   1:  PR[GP1:91,1] = PR[GP1:90,1] + 7.172;
   1:  PR[GP1:91,2] = PR[GP1:90,2] + -12.649;
   1:L PR[91] 10mm/sec CNT100;
   1:  PR[GP1:91,1] = PR[GP1:90,1] + 9.973;
   1:  PR[GP1:91,2] = PR[GP1:90,2] + -18.239;
   1:L PR[91] 10mm/sec CNT100;
   1:  PR[GP1:91,1] = PR[GP1:90,1] + 13.438;
   1:  PR[GP1:91,2] = PR[GP1:90,2] + -22.690;
   1:L PR[91] 10mm/sec CNT100;
   1:  PR[GP1:91,1] = PR[GP1:90,1] + 17.099;
   1:  PR[GP1:91,2] = PR[GP1:90,2] + -26.371;
   1:L PR[91] 10mm/sec CNT100;
   1:  PR[GP1:91,1] = PR[GP1:90,1] + 22.911;
   1:  PR[GP1:91,2] = PR[GP1:90,2] + -30.145;
   1:L PR[91] 10mm/sec CNT100;
   1:  PR[GP1:91,1] = PR[GP1:90,1] + 26.457;
   1:  PR[GP1:91,2] = PR[GP1:90,2] + -31.958;
   1:L PR[91] 10mm/sec CNT100;
   1:  PR[GP1:91,1] = PR[GP1:90,1] + 34.555;
   1:  PR[GP1:91,2] = PR[GP1:90,2] + -33.996;
   1:L PR[91] 10mm/sec CNT100;
   1:  PR[GP1:91,1] = PR[GP1:90,1] + 37.222;
   1:  PR[GP1:91,2] = PR[GP1:90,2] + -34.430;
   1:L PR[91] 10mm/sec CNT100;
   1:  PR[GP1:91,1] = PR[GP1:90,1] + 46.851;
   1:  PR[GP1:91,2] = PR[GP1:90,2] + -33.641;
   1:L PR[91] 10mm/sec CNT100;
   1:  PR[GP1:91,1] = PR[GP1:90,1] + 48.358;
   1:  PR[GP1:91,2] = PR[GP1:90,2] + -33.412;
   1:L PR[91] 10mm/sec CNT100;
   1:  PR[GP1:91,1] = PR[GP1:90,1] + 58.186;
   1:  PR[GP1:91,2] = PR[GP1:90,2] + -29.141;
   1:L PR[91] 10mm/sec CNT100;
   1:  PR[GP1:91,1] = PR[GP1:90,1] + 58.697;
   1:  PR[GP1:91,2] = PR[GP1:90,2] + -28.887;
   1:L PR[91] 10mm/sec CNT100;
   1:  PR[GP1:91,1] = PR[GP1:90,1] + 67.093;
   1:  PR[GP1:91,2] = PR[GP1:90,2] + -21.226;
   1:L PR[91] 10mm/sec CNT100;
   1:  PR[GP1:91,1] = PR[GP1:90,1] + 72.535;
   1:  PR[GP1:91,2] = PR[GP1:90,2] + -11.242;
   1:L PR[91] 10mm/sec CNT100;
   1:  PR[GP1:91,1] = PR[GP1:90,1] + 72.559;
   1:  PR[GP1:91,2] = PR[GP1:90,2] + -11.160;
   1:L PR[91] 10mm/sec CNT100;
   1:  PR[GP1:91,1] = PR[GP1:90,1] + 72.575;
   1:  PR[GP1:91,2] = PR[GP1:90,2] + -10.988;
   1:L PR[91] 10mm/sec CNT100;
   1:  PR[GP1:91,1] = PR[GP1:90,1] + 74.410;
   1:  PR[GP1:91,2] = PR[GP1:90,2] + 0.017;
   1:L PR[91] 10mm/sec CNT100;
   1:  PR[GP1:91,1] = PR[GP1:90,1] + 74.379;
   1:  PR[GP1:91,2] = PR[GP1:90,2] + 0.350;
   1:L PR[91] 10mm/sec CNT100;
   1:  PR[GP1:91,1] = PR[GP1:90,1] + 72.565;
   1:  PR[GP1:91,2] = PR[GP1:90,2] + 11.130;
   1:L PR[91] 10mm/sec CNT100;
   1:  PR[GP1:91,1] = PR[GP1:90,1] + 72.535;
   1:  PR[GP1:91,2] = PR[GP1:90,2] + 11.234;
   1:L PR[91] 10mm/sec CNT100;
   1:  PR[GP1:91,1] = PR[GP1:90,1] + 67.091;
   1:  PR[GP1:91,2] = PR[GP1:90,2] + 21.219;
   1:L PR[91] 10mm/sec CNT100;
   1:  PR[GP1:91,1] = PR[GP1:90,1] + 58.697;
   1:  PR[GP1:91,2] = PR[GP1:90,2] + 28.878;
   1:L PR[91] 10mm/sec CNT100;
   1:  PR[GP1:91,1] = PR[GP1:90,1] + 58.186;
   1:  PR[GP1:91,2] = PR[GP1:90,2] + 29.133;
   1:L PR[91] 10mm/sec CNT100;
   1:  PR[GP1:91,1] = PR[GP1:90,1] + 48.358;
   1:  PR[GP1:91,2] = PR[GP1:90,2] + 33.403;
   1:L PR[91] 10mm/sec CNT100;
   1:  PR[GP1:91,1] = PR[GP1:90,1] + 46.851;
   1:  PR[GP1:91,2] = PR[GP1:90,2] + 33.632;
   1:L PR[91] 10mm/sec CNT100;
   1:  PR[GP1:91,1] = PR[GP1:90,1] + 37.222;
   1:  PR[GP1:91,2] = PR[GP1:90,2] + 34.421;
   1:L PR[91] 10mm/sec CNT100;
   1:  PR[GP1:91,1] = PR[GP1:90,1] + 34.555;
   1:  PR[GP1:91,2] = PR[GP1:90,2] + 33.987;
   1:L PR[91] 10mm/sec CNT100;
   1:  PR[GP1:91,1] = PR[GP1:90,1] + 26.457;
   1:  PR[GP1:91,2] = PR[GP1:90,2] + 31.949;
   1:L PR[91] 10mm/sec CNT100;
   1:  PR[GP1:91,1] = PR[GP1:90,1] + 22.911;
   1:  PR[GP1:91,2] = PR[GP1:90,2] + 30.136;
   1:L PR[91] 10mm/sec CNT100;
   1:  PR[GP1:91,1] = PR[GP1:90,1] + 17.099;
   1:  PR[GP1:91,2] = PR[GP1:90,2] + 26.362;
   1:L PR[91] 10mm/sec CNT100;
   1:  PR[GP1:91,1] = PR[GP1:90,1] + 13.438;
   1:  PR[GP1:91,2] = PR[GP1:90,2] + 22.681;
   1:L PR[91] 10mm/sec CNT100;
   1:  PR[GP1:91,1] = PR[GP1:90,1] + 9.973;
   1:  PR[GP1:91,2] = PR[GP1:90,2] + 18.230;
   1:L PR[91] 10mm/sec CNT100;
   1:  PR[GP1:91,1] = PR[GP1:90,1] + 7.168;
   1:  PR[GP1:91,2] = PR[GP1:90,2] + 12.628;
   1:L PR[91] 10mm/sec CNT100;
   1:  PR[GP1:91,1] = PR[GP1:90,1] + 5.691;
   1:  PR[GP1:91,2] = PR[GP1:90,2] + 8.281;
   1:L PR[91] 10mm/sec CNT100;
   1:  PR[GP1:91,1] = PR[GP1:90,1] + 5.052;
   1:  PR[GP1:91,2] = PR[GP1:90,2] + 6.468;
   1:L PR[91] 10mm/sec CNT100;
   1:  PR[GP1:91,1] = PR[GP1:90,1] + 4.191;
   1:  PR[GP1:91,2] = PR[GP1:90,2] + 5.426;
   1:L PR[91] 10mm/sec CNT100;
   1:  PR[GP1:91,1] = PR[GP1:90,1] + 2.887;
   1:  PR[GP1:91,2] = PR[GP1:90,2] + 4.007;
   1:L PR[91] 10mm/sec CNT100;
   1:  PR[GP1:91,1] = PR[GP1:90,1] + 2.240;
   1:  PR[GP1:91,2] = PR[GP1:90,2] + 3.649;
   1:L PR[91] 10mm/sec CNT100;
   1:  PR[GP1:91,1] = PR[GP1:90,1] + 0.884;
   1:  PR[GP1:91,2] = PR[GP1:90,2] + 4.821;
   1:  PR[GP1:91,3] = PR[GP1:90,3] + 21.280;
   1:L PR[91] 10mm/sec CNT100;
   1:  PR[GP1:91,1] = PR[GP1:90,1] + -1.866;
   1:  PR[GP1:91,2] = PR[GP1:90,2] + 5.029;
   1:L PR[91] 10mm/sec CNT100;
   1:  PR[GP1:91,1] = PR[GP1:90,1] + -2.248;
   1:  PR[GP1:91,2] = PR[GP1:90,2] + 5.297;
   1:L PR[91] 10mm/sec CNT100;
   1:  PR[GP1:91,1] = PR[GP1:90,1] + -3.405;
   1:  PR[GP1:91,2] = PR[GP1:90,2] + 6.715;
   1:L PR[91] 10mm/sec CNT100;
   1:  PR[GP1:91,1] = PR[GP1:90,1] + -4.805;
   1:  PR[GP1:91,2] = PR[GP1:90,2] + 9.191;
   1:L PR[91] 10mm/sec CNT100;
   1:  PR[GP1:91,1] = PR[GP1:90,1] + -5.571;
   1:  PR[GP1:91,2] = PR[GP1:90,2] + 11.449;
   1:L PR[91] 10mm/sec CNT100;
   1:  PR[GP1:91,1] = PR[GP1:90,1] + -9.332;
   1:  PR[GP1:91,2] = PR[GP1:90,2] + 18.969;
   1:L PR[91] 10mm/sec CNT100;
   1:  PR[GP1:91,1] = PR[GP1:90,1] + -11.484;
   1:  PR[GP1:91,2] = PR[GP1:90,2] + 21.732;
   1:L PR[91] 10mm/sec CNT100;
   1:  PR[GP1:91,1] = PR[GP1:90,1] + -16.563;
   1:  PR[GP1:91,2] = PR[GP1:90,2] + 26.824;
   1:L PR[91] 10mm/sec CNT100;
   1:  PR[GP1:91,1] = PR[GP1:90,1] + -20.680;
   1:  PR[GP1:91,2] = PR[GP1:90,2] + 29.498;
   1:L PR[91] 10mm/sec CNT100;
   1:  PR[GP1:91,1] = PR[GP1:90,1] + -25.923;
   1:  PR[GP1:91,2] = PR[GP1:90,2] + 32.179;
   1:L PR[91] 10mm/sec CNT100;
   1:  PR[GP1:91,1] = PR[GP1:90,1] + -32.191;
   1:  PR[GP1:91,2] = PR[GP1:90,2] + 33.756;
   1:L PR[91] 10mm/sec CNT100;
   1:  PR[GP1:91,1] = PR[GP1:90,1] + -36.623;
   1:  PR[GP1:91,2] = PR[GP1:90,2] + 34.474;
   1:L PR[91] 10mm/sec CNT100;
   1:  PR[GP1:91,1] = PR[GP1:90,1] + -44.511;
   1:  PR[GP1:91,2] = PR[GP1:90,2] + 33.827;
   1:L PR[91] 10mm/sec CNT100;
   1:  PR[GP1:91,1] = PR[GP1:90,1] + -47.660;
   1:  PR[GP1:91,2] = PR[GP1:90,2] + 33.349;
   1:L PR[91] 10mm/sec CNT100;
   1:  PR[GP1:91,1] = PR[GP1:90,1] + -56.007;
   1:  PR[GP1:91,2] = PR[GP1:90,2] + 29.720;
   1:L PR[91] 10mm/sec CNT100;
   1:  PR[GP1:91,1] = PR[GP1:90,1] + -57.896;
   1:  PR[GP1:91,2] = PR[GP1:90,2] + 28.777;
   1:L PR[91] 10mm/sec CNT100;
   1:  PR[GP1:91,1] = PR[GP1:90,1] + -65.248;
   1:  PR[GP1:91,2] = PR[GP1:90,2] + 22.071;
   1:L PR[91] 10mm/sec CNT100;
   1:  PR[GP1:91,1] = PR[GP1:90,1] + -66.199;
   1:  PR[GP1:91,2] = PR[GP1:90,2] + 21.135;
   1:L PR[91] 10mm/sec CNT100;
   1:  PR[GP1:91,1] = PR[GP1:90,1] + -71.212;
   1:  PR[GP1:91,2] = PR[GP1:90,2] + 11.956;
   1:L PR[91] 10mm/sec CNT100;
   1:  PR[GP1:91,1] = PR[GP1:90,1] + -71.611;
   1:  PR[GP1:91,2] = PR[GP1:90,2] + 11.183;
   1:L PR[91] 10mm/sec CNT100;
   1:  PR[GP1:91,1] = PR[GP1:90,1] + -73.500;
   1:  PR[GP1:91,2] = PR[GP1:90,2] + -0.004;
   1:L PR[91] 10mm/sec CNT100;
   1:  PR[GP1:91,1] = PR[GP1:90,1] + -71.736;
   1:  PR[GP1:91,2] = PR[GP1:90,2] + -10.406;
   1:L PR[91] 10mm/sec CNT100;
   1:  PR[GP1:91,1] = PR[GP1:90,1] + -71.610;
   1:  PR[GP1:91,2] = PR[GP1:90,2] + -11.194;
   1:L PR[91] 10mm/sec CNT100;
   1:  PR[GP1:91,1] = PR[GP1:90,1] + -71.212;
   1:  PR[GP1:91,2] = PR[GP1:90,2] + -11.965;
   1:L PR[91] 10mm/sec CNT100;
   1:  PR[GP1:91,1] = PR[GP1:90,1] + -66.199;
   1:  PR[GP1:91,2] = PR[GP1:90,2] + -21.144;
   1:L PR[91] 10mm/sec CNT100;
   1:  PR[GP1:91,1] = PR[GP1:90,1] + -65.248;
   1:  PR[GP1:91,2] = PR[GP1:90,2] + -22.080;
   1:L PR[91] 10mm/sec CNT100;
   1:  PR[GP1:91,1] = PR[GP1:90,1] + -57.896;
   1:  PR[GP1:91,2] = PR[GP1:90,2] + -28.786;
   1:L PR[91] 10mm/sec CNT100;
   1:  PR[GP1:91,1] = PR[GP1:90,1] + -56.007;
   1:  PR[GP1:91,2] = PR[GP1:90,2] + -29.729;
   1:L PR[91] 10mm/sec CNT100;
   1:  PR[GP1:91,1] = PR[GP1:90,1] + -47.660;
   1:  PR[GP1:91,2] = PR[GP1:90,2] + -33.358;
   1:L PR[91] 10mm/sec CNT100;
   1:  PR[GP1:91,1] = PR[GP1:90,1] + -44.511;
   1:  PR[GP1:91,2] = PR[GP1:90,2] + -33.836;
   1:L PR[91] 10mm/sec CNT100;
   1:  PR[GP1:91,1] = PR[GP1:90,1] + -36.623;
   1:  PR[GP1:91,2] = PR[GP1:90,2] + -34.483;
   1:L PR[91] 10mm/sec CNT100;
   1:  PR[GP1:91,1] = PR[GP1:90,1] + -32.191;
   1:  PR[GP1:91,2] = PR[GP1:90,2] + -33.765;
   1:L PR[91] 10mm/sec CNT100;
   1:  PR[GP1:91,1] = PR[GP1:90,1] + -25.924;
   1:  PR[GP1:91,2] = PR[GP1:90,2] + -32.188;
   1:L PR[91] 10mm/sec CNT100;
   1:  PR[GP1:91,1] = PR[GP1:90,1] + -20.680;
   1:  PR[GP1:91,2] = PR[GP1:90,2] + -29.507;
   1:L PR[91] 10mm/sec CNT100;
   1:  PR[GP1:91,1] = PR[GP1:90,1] + -16.563;
   1:  PR[GP1:91,2] = PR[GP1:90,2] + -26.833;
   1:L PR[91] 10mm/sec CNT100;
   1:  PR[GP1:91,1] = PR[GP1:90,1] + -11.484;
   1:  PR[GP1:91,2] = PR[GP1:90,2] + -21.741;
   1:L PR[91] 10mm/sec CNT100;
   1:  PR[GP1:91,1] = PR[GP1:90,1] + -9.332;
   1:  PR[GP1:91,2] = PR[GP1:90,2] + -18.977;
   1:L PR[91] 10mm/sec CNT100;
   1:  PR[GP1:91,1] = PR[GP1:90,1] + -5.576;
   1:  PR[GP1:91,2] = PR[GP1:90,2] + -11.474;
   1:L PR[91] 10mm/sec CNT100;
   1:  PR[GP1:91,1] = PR[GP1:90,1] + -4.308;
   1:  PR[GP1:91,2] = PR[GP1:90,2] + -7.786;
   1:L PR[91] 10mm/sec CNT100;
   1:  PR[GP1:91,1] = PR[GP1:90,1] + -3.131;
   1:  PR[GP1:91,2] = PR[GP1:90,2] + -6.484;
   1:L PR[91] 10mm/sec CNT100;
   1:  PR[GP1:91,1] = PR[GP1:90,1] + -2.802;
   1:  PR[GP1:91,2] = PR[GP1:90,2] + -6.283;
   1:L PR[91] 10mm/sec CNT100;
   1:  PR[GP1:91,1] = PR[GP1:90,1] + -1.567;
   1:  PR[GP1:91,2] = PR[GP1:90,2] + -4.807;
   1:L PR[91] 10mm/sec CNT100;
   1:  PR[GP1:91,1] = PR[GP1:90,1] + 1.456;
   1:  PR[GP1:91,2] = PR[GP1:90,2] + -5.040;
   1:L PR[91] 10mm/sec CNT100;
   1:  PR[GP1:91,1] = PR[GP1:90,1] + 1.588;
   1:  PR[GP1:91,2] = PR[GP1:90,2] + -5.147;
   1:L PR[91] 10mm/sec CNT100;
   1:  PR[GP1:91,1] = PR[GP1:90,1] + 2.989;
   1:  PR[GP1:91,2] = PR[GP1:90,2] + -5.133;
   1:L PR[91] 10mm/sec CNT100;
   1:  PR[GP1:91,1] = PR[GP1:90,1] + 4.319;
   1:  PR[GP1:91,2] = PR[GP1:90,2] + -7.663;
   1:L PR[91] 10mm/sec CNT100;
   1:  PR[GP1:91,1] = PR[GP1:90,1] + 5.601;
   1:  PR[GP1:91,2] = PR[GP1:90,2] + -9.140;
   1:L PR[91] 10mm/sec CNT100;
   1:  PR[GP1:91,1] = PR[GP1:90,1] + 6.392;
   1:  PR[GP1:91,2] = PR[GP1:90,2] + -11.470;
   1:L PR[91] 10mm/sec CNT100;
   1:  PR[GP1:91,1] = PR[GP1:90,1] + 10.145;
   1:  PR[GP1:91,2] = PR[GP1:90,2] + -18.959;
   1:L PR[91] 10mm/sec CNT100;
   1:  PR[GP1:91,1] = PR[GP1:90,1] + 12.297;
   1:  PR[GP1:91,2] = PR[GP1:90,2] + -21.723;
   1:L PR[91] 10mm/sec CNT100;
   1:  PR[GP1:91,1] = PR[GP1:90,1] + 17.376;
   1:  PR[GP1:91,2] = PR[GP1:90,2] + -26.830;
   1:L PR[91] 10mm/sec CNT100;
   1:  PR[GP1:91,1] = PR[GP1:90,1] + 21.491;
   1:  PR[GP1:91,2] = PR[GP1:90,2] + -29.502;
   1:L PR[91] 10mm/sec CNT100;
   1:  PR[GP1:91,1] = PR[GP1:90,1] + 26.737;
   1:  PR[GP1:91,2] = PR[GP1:90,2] + -32.185;
   1:L PR[91] 10mm/sec CNT100;
   1:  PR[GP1:91,1] = PR[GP1:90,1] + 33.004;
   1:  PR[GP1:91,2] = PR[GP1:90,2] + -33.762;
   1:L PR[91] 10mm/sec CNT100;
   1:  PR[GP1:91,1] = PR[GP1:90,1] + 37.438;
   1:  PR[GP1:91,2] = PR[GP1:90,2] + -34.483;
   1:L PR[91] 10mm/sec CNT100;
   1:  PR[GP1:91,1] = PR[GP1:90,1] + 45.326;
   1:  PR[GP1:91,2] = PR[GP1:90,2] + -33.836;
   1:L PR[91] 10mm/sec CNT100;
   1:  PR[GP1:91,1] = PR[GP1:90,1] + 48.477;
   1:  PR[GP1:91,2] = PR[GP1:90,2] + -33.358;
   1:L PR[91] 10mm/sec CNT100;
   1:  PR[GP1:91,1] = PR[GP1:90,1] + 56.825;
   1:  PR[GP1:91,2] = PR[GP1:90,2] + -29.731;
   1:L PR[91] 10mm/sec CNT100;
   1:  PR[GP1:91,1] = PR[GP1:90,1] + 58.715;
   1:  PR[GP1:91,2] = PR[GP1:90,2] + -28.789;
   1:L PR[91] 10mm/sec CNT100;
   1:  PR[GP1:91,1] = PR[GP1:90,1] + 66.067;
   1:  PR[GP1:91,2] = PR[GP1:90,2] + -22.080;
   1:L PR[91] 10mm/sec CNT100;
   1:  PR[GP1:91,1] = PR[GP1:90,1] + 67.019;
   1:  PR[GP1:91,2] = PR[GP1:90,2] + -21.142;
   1:L PR[91] 10mm/sec CNT100;
   1:  PR[GP1:91,1] = PR[GP1:90,1] + 72.032;
   1:  PR[GP1:91,2] = PR[GP1:90,2] + -11.969;
   1:L PR[91] 10mm/sec CNT100;
   1:  PR[GP1:91,1] = PR[GP1:90,1] + 72.432;
   1:  PR[GP1:91,2] = PR[GP1:90,2] + -11.197;
   1:L PR[91] 10mm/sec CNT100;
   1:  PR[GP1:91,1] = PR[GP1:90,1] + 74.321;
   1:  PR[GP1:91,2] = PR[GP1:90,2] + -0.004;
   1:L PR[91] 10mm/sec CNT100;
   1:  PR[GP1:91,1] = PR[GP1:90,1] + 72.432;
   1:  PR[GP1:91,2] = PR[GP1:90,2] + 11.188;
   1:L PR[91] 10mm/sec CNT100;
   1:  PR[GP1:91,1] = PR[GP1:90,1] + 72.032;
   1:  PR[GP1:91,2] = PR[GP1:90,2] + 11.960;
   1:L PR[91] 10mm/sec CNT100;
   1:  PR[GP1:91,1] = PR[GP1:90,1] + 67.019;
   1:  PR[GP1:91,2] = PR[GP1:90,2] + 21.133;
   1:L PR[91] 10mm/sec CNT100;
   1:  PR[GP1:91,1] = PR[GP1:90,1] + 66.067;
   1:  PR[GP1:91,2] = PR[GP1:90,2] + 22.071;
   1:L PR[91] 10mm/sec CNT100;
   1:  PR[GP1:91,1] = PR[GP1:90,1] + 58.715;
   1:  PR[GP1:91,2] = PR[GP1:90,2] + 28.780;
   1:L PR[91] 10mm/sec CNT100;
   1:  PR[GP1:91,1] = PR[GP1:90,1] + 56.825;
   1:  PR[GP1:91,2] = PR[GP1:90,2] + 29.722;
   1:L PR[91] 10mm/sec CNT100;
   1:  PR[GP1:91,1] = PR[GP1:90,1] + 48.477;
   1:  PR[GP1:91,2] = PR[GP1:90,2] + 33.349;
   1:L PR[91] 10mm/sec CNT100;
   1:  PR[GP1:91,1] = PR[GP1:90,1] + 45.326;
   1:  PR[GP1:91,2] = PR[GP1:90,2] + 33.828;
   1:L PR[91] 10mm/sec CNT100;
   1:  PR[GP1:91,1] = PR[GP1:90,1] + 37.438;
   1:  PR[GP1:91,2] = PR[GP1:90,2] + 34.474;
   1:L PR[91] 10mm/sec CNT100;
   1:  PR[GP1:91,1] = PR[GP1:90,1] + 33.004;
   1:  PR[GP1:91,2] = PR[GP1:90,2] + 33.753;
   1:L PR[91] 10mm/sec CNT100;
   1:  PR[GP1:91,1] = PR[GP1:90,1] + 26.737;
   1:  PR[GP1:91,2] = PR[GP1:90,2] + 32.176;
   1:L PR[91] 10mm/sec CNT100;
   1:  PR[GP1:91,1] = PR[GP1:90,1] + 21.491;
   1:  PR[GP1:91,2] = PR[GP1:90,2] + 29.494;
   1:L PR[91] 10mm/sec CNT100;
   1:  PR[GP1:91,1] = PR[GP1:90,1] + 17.375;
   1:  PR[GP1:91,2] = PR[GP1:90,2] + 26.821;
   1:L PR[91] 10mm/sec CNT100;
   1:  PR[GP1:91,1] = PR[GP1:90,1] + 12.297;
   1:  PR[GP1:91,2] = PR[GP1:90,2] + 21.714;
   1:L PR[91] 10mm/sec CNT100;
   1:  PR[GP1:91,1] = PR[GP1:90,1] + 10.145;
   1:  PR[GP1:91,2] = PR[GP1:90,2] + 18.950;
   1:L PR[91] 10mm/sec CNT100;
   1:  PR[GP1:91,1] = PR[GP1:90,1] + 6.385;
   1:  PR[GP1:91,2] = PR[GP1:90,2] + 11.443;
   1:L PR[91] 10mm/sec CNT100;
   1:  PR[GP1:91,1] = PR[GP1:90,1] + 5.125;
   1:  PR[GP1:91,2] = PR[GP1:90,2] + 7.774;
   1:L PR[91] 10mm/sec CNT100;
   1:  PR[GP1:91,1] = PR[GP1:90,1] + 3.922;
   1:  PR[GP1:91,2] = PR[GP1:90,2] + 6.317;
   1:L PR[91] 10mm/sec CNT100;
   1:  PR[GP1:91,1] = PR[GP1:90,1] + 2.826;
   1:  PR[GP1:91,2] = PR[GP1:90,2] + 5.125;
   1:L PR[91] 10mm/sec CNT100;
   1:  PR[GP1:91,1] = PR[GP1:90,1] + 2.251;
   1:  PR[GP1:91,2] = PR[GP1:90,2] + 4.806;
   1:L PR[91] 10mm/sec CNT100;
   1:  PR[GP1:91,1] = PR[GP1:90,1] + 0.410;
   1:  PR[GP1:91,2] = PR[GP1:90,2] + 5.983;
   1:  PR[GP1:91,3] = PR[GP1:90,3] + 22.610;
   1:L PR[91] 10mm/sec CNT100;
   1:  PR[GP1:91,1] = PR[GP1:90,1] + -1.815;
   1:  PR[GP1:91,2] = PR[GP1:90,2] + 6.152;
   1:L PR[91] 10mm/sec CNT100;
   1:  PR[GP1:91,1] = PR[GP1:90,1] + -2.161;
   1:  PR[GP1:91,2] = PR[GP1:90,2] + 6.394;
   1:L PR[91] 10mm/sec CNT100;
   1:  PR[GP1:91,1] = PR[GP1:90,1] + -3.724;
   1:  PR[GP1:91,2] = PR[GP1:90,2] + 8.310;
   1:L PR[91] 10mm/sec CNT100;
   1:  PR[GP1:91,1] = PR[GP1:90,1] + -4.752;
   1:  PR[GP1:91,2] = PR[GP1:90,2] + 10.152;
   1:L PR[91] 10mm/sec CNT100;
   1:  PR[GP1:91,1] = PR[GP1:90,1] + -4.791;
   1:  PR[GP1:91,2] = PR[GP1:90,2] + 10.265;
   1:L PR[91] 10mm/sec CNT100;
   1:  PR[GP1:91,1] = PR[GP1:90,1] + -9.505;
   1:  PR[GP1:91,2] = PR[GP1:90,2] + 19.692;
   1:L PR[91] 10mm/sec CNT100;
   1:  PR[GP1:91,1] = PR[GP1:90,1] + -10.345;
   1:  PR[GP1:91,2] = PR[GP1:90,2] + 20.769;
   1:L PR[91] 10mm/sec CNT100;
   1:  PR[GP1:91,1] = PR[GP1:90,1] + -16.841;
   1:  PR[GP1:91,2] = PR[GP1:90,2] + 27.284;
   1:L PR[91] 10mm/sec CNT100;
   1:  PR[GP1:91,1] = PR[GP1:90,1] + -19.262;
   1:  PR[GP1:91,2] = PR[GP1:90,2] + 28.856;
   1:L PR[91] 10mm/sec CNT100;
   1:  PR[GP1:91,1] = PR[GP1:90,1] + -26.205;
   1:  PR[GP1:91,2] = PR[GP1:90,2] + 32.407;
   1:L PR[91] 10mm/sec CNT100;
   1:  PR[GP1:91,1] = PR[GP1:90,1] + -30.643;
   1:  PR[GP1:91,2] = PR[GP1:90,2] + 33.523;
   1:L PR[91] 10mm/sec CNT100;
   1:  PR[GP1:91,1] = PR[GP1:90,1] + -36.840;
   1:  PR[GP1:91,2] = PR[GP1:90,2] + 34.527;
   1:L PR[91] 10mm/sec CNT100;
   1:  PR[GP1:91,1] = PR[GP1:90,1] + -42.988;
   1:  PR[GP1:91,2] = PR[GP1:90,2] + 34.023;
   1:L PR[91] 10mm/sec CNT100;
   1:  PR[GP1:91,1] = PR[GP1:90,1] + -47.779;
   1:  PR[GP1:91,2] = PR[GP1:90,2] + 33.295;
   1:L PR[91] 10mm/sec CNT100;
   1:  PR[GP1:91,1] = PR[GP1:90,1] + -54.648;
   1:  PR[GP1:91,2] = PR[GP1:90,2] + 30.310;
   1:L PR[91] 10mm/sec CNT100;
   1:  PR[GP1:91,1] = PR[GP1:90,1] + -57.914;
   1:  PR[GP1:91,2] = PR[GP1:90,2] + 28.679;
   1:L PR[91] 10mm/sec CNT100;
   1:  PR[GP1:91,1] = PR[GP1:90,1] + -64.160;
   1:  PR[GP1:91,2] = PR[GP1:90,2] + 22.982;
   1:L PR[91] 10mm/sec CNT100;
   1:  PR[GP1:91,1] = PR[GP1:90,1] + -66.132;
   1:  PR[GP1:91,2] = PR[GP1:90,2] + 21.041;
   1:L PR[91] 10mm/sec CNT100;
   1:  PR[GP1:91,1] = PR[GP1:90,1] + -70.470;
   1:  PR[GP1:91,2] = PR[GP1:90,2] + 13.096;
   1:L PR[91] 10mm/sec CNT100;
   1:  PR[GP1:91,1] = PR[GP1:90,1] + -71.488;
   1:  PR[GP1:91,2] = PR[GP1:90,2] + 11.127;
   1:L PR[91] 10mm/sec CNT100;
   1:  PR[GP1:91,1] = PR[GP1:90,1] + -73.081;
   1:  PR[GP1:91,2] = PR[GP1:90,2] + 1.714;
   1:L PR[91] 10mm/sec CNT100;
   1:  PR[GP1:91,1] = PR[GP1:90,1] + -73.356;
   1:  PR[GP1:91,2] = PR[GP1:90,2] + -0.002;
   1:L PR[91] 10mm/sec CNT100;
   1:  PR[GP1:91,1] = PR[GP1:90,1] + -71.808;
   1:  PR[GP1:91,2] = PR[GP1:90,2] + -9.130;
   1:L PR[91] 10mm/sec CNT100;
   1:  PR[GP1:91,1] = PR[GP1:90,1] + -71.486;
   1:  PR[GP1:91,2] = PR[GP1:90,2] + -11.139;
   1:L PR[91] 10mm/sec CNT100;
   1:  PR[GP1:91,1] = PR[GP1:90,1] + -70.470;
   1:  PR[GP1:91,2] = PR[GP1:90,2] + -13.105;
   1:L PR[91] 10mm/sec CNT100;
   1:  PR[GP1:91,1] = PR[GP1:90,1] + -66.132;
   1:  PR[GP1:91,2] = PR[GP1:90,2] + -21.050;
   1:L PR[91] 10mm/sec CNT100;
   1:  PR[GP1:91,1] = PR[GP1:90,1] + -64.159;
   1:  PR[GP1:91,2] = PR[GP1:90,2] + -22.991;
   1:L PR[91] 10mm/sec CNT100;
   1:  PR[GP1:91,1] = PR[GP1:90,1] + -57.914;
   1:  PR[GP1:91,2] = PR[GP1:90,2] + -28.688;
   1:L PR[91] 10mm/sec CNT100;
   1:  PR[GP1:91,1] = PR[GP1:90,1] + -54.648;
   1:  PR[GP1:91,2] = PR[GP1:90,2] + -30.319;
   1:L PR[91] 10mm/sec CNT100;
   1:  PR[GP1:91,1] = PR[GP1:90,1] + -47.779;
   1:  PR[GP1:91,2] = PR[GP1:90,2] + -33.304;
   1:L PR[91] 10mm/sec CNT100;
   1:  PR[GP1:91,1] = PR[GP1:90,1] + -42.988;
   1:  PR[GP1:91,2] = PR[GP1:90,2] + -34.032;
   1:L PR[91] 10mm/sec CNT100;
   1:  PR[GP1:91,1] = PR[GP1:90,1] + -36.840;
   1:  PR[GP1:91,2] = PR[GP1:90,2] + -34.536;
   1:L PR[91] 10mm/sec CNT100;
   1:  PR[GP1:91,1] = PR[GP1:90,1] + -30.643;
   1:  PR[GP1:91,2] = PR[GP1:90,2] + -33.532;
   1:L PR[91] 10mm/sec CNT100;
   1:  PR[GP1:91,1] = PR[GP1:90,1] + -26.205;
   1:  PR[GP1:91,2] = PR[GP1:90,2] + -32.415;
   1:L PR[91] 10mm/sec CNT100;
   1:  PR[GP1:91,1] = PR[GP1:90,1] + -19.262;
   1:  PR[GP1:91,2] = PR[GP1:90,2] + -28.865;
   1:L PR[91] 10mm/sec CNT100;
   1:  PR[GP1:91,1] = PR[GP1:90,1] + -16.841;
   1:  PR[GP1:91,2] = PR[GP1:90,2] + -27.293;
   1:L PR[91] 10mm/sec CNT100;
   1:  PR[GP1:91,1] = PR[GP1:90,1] + -10.345;
   1:  PR[GP1:91,2] = PR[GP1:90,2] + -20.778;
   1:L PR[91] 10mm/sec CNT100;
   1:  PR[GP1:91,1] = PR[GP1:90,1] + -9.505;
   1:  PR[GP1:91,2] = PR[GP1:90,2] + -19.701;
   1:L PR[91] 10mm/sec CNT100;
   1:  PR[GP1:91,1] = PR[GP1:90,1] + -4.797;
   1:  PR[GP1:91,2] = PR[GP1:90,2] + -10.293;
   1:L PR[91] 10mm/sec CNT100;
   1:  PR[GP1:91,1] = PR[GP1:90,1] + -4.382;
   1:  PR[GP1:91,2] = PR[GP1:90,2] + -9.094;
   1:L PR[91] 10mm/sec CNT100;
   1:  PR[GP1:91,1] = PR[GP1:90,1] + -3.503;
   1:  PR[GP1:91,2] = PR[GP1:90,2] + -8.122;
   1:L PR[91] 10mm/sec CNT100;
   1:  PR[GP1:91,1] = PR[GP1:90,1] + -3.272;
   1:  PR[GP1:91,2] = PR[GP1:90,2] + -7.981;
   1:L PR[91] 10mm/sec CNT100;
   1:  PR[GP1:91,1] = PR[GP1:90,1] + -1.588;
   1:  PR[GP1:91,2] = PR[GP1:90,2] + -5.970;
   1:L PR[91] 10mm/sec CNT100;
   1:  PR[GP1:91,1] = PR[GP1:90,1] + 0.917;
   1:  PR[GP1:91,2] = PR[GP1:90,2] + -6.163;
   1:L PR[91] 10mm/sec CNT100;
   1:  PR[GP1:91,1] = PR[GP1:90,1] + 1.018;
   1:  PR[GP1:91,2] = PR[GP1:90,2] + -6.244;
   1:L PR[91] 10mm/sec CNT100;
   1:  PR[GP1:91,1] = PR[GP1:90,1] + 2.892;
   1:  PR[GP1:91,2] = PR[GP1:90,2] + -6.225;
   1:L PR[91] 10mm/sec CNT100;
   1:  PR[GP1:91,1] = PR[GP1:90,1] + 3.978;
   1:  PR[GP1:91,2] = PR[GP1:90,2] + -8.293;
   1:L PR[91] 10mm/sec CNT100;
   1:  PR[GP1:91,1] = PR[GP1:90,1] + 5.547;
   1:  PR[GP1:91,2] = PR[GP1:90,2] + -10.099;
   1:L PR[91] 10mm/sec CNT100;
   1:  PR[GP1:91,1] = PR[GP1:90,1] + 5.611;
   1:  PR[GP1:91,2] = PR[GP1:90,2] + -10.290;
   1:L PR[91] 10mm/sec CNT100;
   1:  PR[GP1:91,1] = PR[GP1:90,1] + 10.317;
   1:  PR[GP1:91,2] = PR[GP1:90,2] + -19.679;
   1:L PR[91] 10mm/sec CNT100;
   1:  PR[GP1:91,1] = PR[GP1:90,1] + 11.155;
   1:  PR[GP1:91,2] = PR[GP1:90,2] + -20.756;
   1:L PR[91] 10mm/sec CNT100;
   1:  PR[GP1:91,1] = PR[GP1:90,1] + 17.652;
   1:  PR[GP1:91,2] = PR[GP1:90,2] + -27.289;
   1:L PR[91] 10mm/sec CNT100;
   1:  PR[GP1:91,1] = PR[GP1:90,1] + 20.071;
   1:  PR[GP1:91,2] = PR[GP1:90,2] + -28.860;
   1:L PR[91] 10mm/sec CNT100;
   1:  PR[GP1:91,1] = PR[GP1:90,1] + 27.017;
   1:  PR[GP1:91,2] = PR[GP1:90,2] + -32.411;
   1:L PR[91] 10mm/sec CNT100;
   1:  PR[GP1:91,1] = PR[GP1:90,1] + 31.454;
   1:  PR[GP1:91,2] = PR[GP1:90,2] + -33.528;
   1:L PR[91] 10mm/sec CNT100;
   1:  PR[GP1:91,1] = PR[GP1:90,1] + 37.654;
   1:  PR[GP1:91,2] = PR[GP1:90,2] + -34.536;
   1:L PR[91] 10mm/sec CNT100;
   1:  PR[GP1:91,1] = PR[GP1:90,1] + 43.802;
   1:  PR[GP1:91,2] = PR[GP1:90,2] + -34.032;
   1:L PR[91] 10mm/sec CNT100;
   1:  PR[GP1:91,1] = PR[GP1:90,1] + 48.596;
   1:  PR[GP1:91,2] = PR[GP1:90,2] + -33.305;
   1:L PR[91] 10mm/sec CNT100;
   1:  PR[GP1:91,1] = PR[GP1:90,1] + 55.464;
   1:  PR[GP1:91,2] = PR[GP1:90,2] + -30.320;
   1:L PR[91] 10mm/sec CNT100;
   1:  PR[GP1:91,1] = PR[GP1:90,1] + 58.732;
   1:  PR[GP1:91,2] = PR[GP1:90,2] + -28.691;
   1:L PR[91] 10mm/sec CNT100;
   1:  PR[GP1:91,1] = PR[GP1:90,1] + 64.978;
   1:  PR[GP1:91,2] = PR[GP1:90,2] + -22.992;
   1:L PR[91] 10mm/sec CNT100;
   1:  PR[GP1:91,1] = PR[GP1:90,1] + 66.951;
   1:  PR[GP1:91,2] = PR[GP1:90,2] + -21.047;
   1:L PR[91] 10mm/sec CNT100;
   1:  PR[GP1:91,1] = PR[GP1:90,1] + 71.290;
   1:  PR[GP1:91,2] = PR[GP1:90,2] + -13.107;
   1:L PR[91] 10mm/sec CNT100;
   1:  PR[GP1:91,1] = PR[GP1:90,1] + 72.308;
   1:  PR[GP1:91,2] = PR[GP1:90,2] + -11.143;
   1:L PR[91] 10mm/sec CNT100;
   1:  PR[GP1:91,1] = PR[GP1:90,1] + 73.902;
   1:  PR[GP1:91,2] = PR[GP1:90,2] + -1.725;
   1:L PR[91] 10mm/sec CNT100;
   1:  PR[GP1:91,1] = PR[GP1:90,1] + 74.177;
   1:  PR[GP1:91,2] = PR[GP1:90,2] + -0.007;
   1:L PR[91] 10mm/sec CNT100;
   1:  PR[GP1:91,1] = PR[GP1:90,1] + 72.628;
   1:  PR[GP1:91,2] = PR[GP1:90,2] + 9.125;
   1:L PR[91] 10mm/sec CNT100;
   1:  PR[GP1:91,1] = PR[GP1:90,1] + 72.307;
   1:  PR[GP1:91,2] = PR[GP1:90,2] + 11.137;
   1:L PR[91] 10mm/sec CNT100;
   1:  PR[GP1:91,1] = PR[GP1:90,1] + 71.290;
   1:  PR[GP1:91,2] = PR[GP1:90,2] + 13.099;
   1:L PR[91] 10mm/sec CNT100;
   1:  PR[GP1:91,1] = PR[GP1:90,1] + 66.951;
   1:  PR[GP1:91,2] = PR[GP1:90,2] + 21.038;
   1:L PR[91] 10mm/sec CNT100;
   1:  PR[GP1:91,1] = PR[GP1:90,1] + 64.978;
   1:  PR[GP1:91,2] = PR[GP1:90,2] + 22.983;
   1:L PR[91] 10mm/sec CNT100;
   1:  PR[GP1:91,1] = PR[GP1:90,1] + 58.732;
   1:  PR[GP1:91,2] = PR[GP1:90,2] + 28.682;
   1:L PR[91] 10mm/sec CNT100;
   1:  PR[GP1:91,1] = PR[GP1:90,1] + 55.464;
   1:  PR[GP1:91,2] = PR[GP1:90,2] + 30.311;
   1:L PR[91] 10mm/sec CNT100;
   1:  PR[GP1:91,1] = PR[GP1:90,1] + 48.596;
   1:  PR[GP1:91,2] = PR[GP1:90,2] + 33.296;
   1:L PR[91] 10mm/sec CNT100;
   1:  PR[GP1:91,1] = PR[GP1:90,1] + 43.802;
   1:  PR[GP1:91,2] = PR[GP1:90,2] + 34.023;
   1:L PR[91] 10mm/sec CNT100;
   1:  PR[GP1:91,1] = PR[GP1:90,1] + 37.654;
   1:  PR[GP1:91,2] = PR[GP1:90,2] + 34.527;
   1:L PR[91] 10mm/sec CNT100;
   1:  PR[GP1:91,1] = PR[GP1:90,1] + 31.454;
   1:  PR[GP1:91,2] = PR[GP1:90,2] + 33.519;
   1:L PR[91] 10mm/sec CNT100;
   1:  PR[GP1:91,1] = PR[GP1:90,1] + 27.017;
   1:  PR[GP1:91,2] = PR[GP1:90,2] + 32.402;
   1:L PR[91] 10mm/sec CNT100;
   1:  PR[GP1:91,1] = PR[GP1:90,1] + 20.071;
   1:  PR[GP1:91,2] = PR[GP1:90,2] + 28.851;
   1:L PR[91] 10mm/sec CNT100;
   1:  PR[GP1:91,1] = PR[GP1:90,1] + 17.652;
   1:  PR[GP1:91,2] = PR[GP1:90,2] + 27.280;
   1:L PR[91] 10mm/sec CNT100;
   1:  PR[GP1:91,1] = PR[GP1:90,1] + 11.155;
   1:  PR[GP1:91,2] = PR[GP1:90,2] + 20.747;
   1:L PR[91] 10mm/sec CNT100;
   1:  PR[GP1:91,1] = PR[GP1:90,1] + 10.317;
   1:  PR[GP1:91,2] = PR[GP1:90,2] + 19.670;
   1:L PR[91] 10mm/sec CNT100;
   1:  PR[GP1:91,1] = PR[GP1:90,1] + 5.604;
   1:  PR[GP1:91,2] = PR[GP1:90,2] + 10.259;
   1:L PR[91] 10mm/sec CNT100;
   1:  PR[GP1:91,1] = PR[GP1:90,1] + 5.196;
   1:  PR[GP1:91,2] = PR[GP1:90,2] + 9.078;
   1:L PR[91] 10mm/sec CNT100;
   1:  PR[GP1:91,1] = PR[GP1:90,1] + 3.653;
   1:  PR[GP1:91,2] = PR[GP1:90,2] + 7.209;
   1:L PR[91] 10mm/sec CNT100;
   1:  PR[GP1:91,1] = PR[GP1:90,1] + 2.765;
   1:  PR[GP1:91,2] = PR[GP1:90,2] + 6.242;
   1:L PR[91] 10mm/sec CNT100;
   1:  PR[GP1:91,1] = PR[GP1:90,1] + 2.261;
   1:  PR[GP1:91,2] = PR[GP1:90,2] + 5.964;
   1:L PR[91] 10mm/sec CNT100;
   1:  PR[GP1:91,1] = PR[GP1:90,1] + -0.065;
   1:  PR[GP1:91,2] = PR[GP1:90,2] + 7.146;
   1:  PR[GP1:91,3] = PR[GP1:90,3] + 23.940;
   1:L PR[91] 10mm/sec CNT100;
   1:  PR[GP1:91,1] = PR[GP1:90,1] + -1.765;
   1:  PR[GP1:91,2] = PR[GP1:90,2] + 7.274;
   1:L PR[91] 10mm/sec CNT100;
   1:  PR[GP1:91,1] = PR[GP1:90,1] + -2.074;
   1:  PR[GP1:91,2] = PR[GP1:90,2] + 7.491;
   1:L PR[91] 10mm/sec CNT100;
   1:  PR[GP1:91,1] = PR[GP1:90,1] + -4.043;
   1:  PR[GP1:91,2] = PR[GP1:90,2] + 9.904;
   1:L PR[91] 10mm/sec CNT100;
   1:  PR[GP1:91,1] = PR[GP1:90,1] + -4.665;
   1:  PR[GP1:91,2] = PR[GP1:90,2] + 11.023;
   1:L PR[91] 10mm/sec CNT100;
   1:  PR[GP1:91,1] = PR[GP1:90,1] + -9.277;
   1:  PR[GP1:91,2] = PR[GP1:90,2] + 19.846;
   1:L PR[91] 10mm/sec CNT100;
   1:  PR[GP1:91,1] = PR[GP1:90,1] + -9.604;
   1:  PR[GP1:91,2] = PR[GP1:90,2] + 20.320;
   1:L PR[91] 10mm/sec CNT100;
   1:  PR[GP1:91,1] = PR[GP1:90,1] + -12.636;
   1:  PR[GP1:91,2] = PR[GP1:90,2] + 23.248;
   1:L PR[91] 10mm/sec CNT100;
   1:  PR[GP1:91,1] = PR[GP1:90,1] + -17.120;
   1:  PR[GP1:91,2] = PR[GP1:90,2] + 27.744;
   1:L PR[91] 10mm/sec CNT100;
   1:  PR[GP1:91,1] = PR[GP1:90,1] + -17.844;
   1:  PR[GP1:91,2] = PR[GP1:90,2] + 28.215;
   1:L PR[91] 10mm/sec CNT100;
   1:  PR[GP1:91,1] = PR[GP1:90,1] + -26.487;
   1:  PR[GP1:91,2] = PR[GP1:90,2] + 32.634;
   1:L PR[91] 10mm/sec CNT100;
   1:  PR[GP1:91,1] = PR[GP1:90,1] + -29.094;
   1:  PR[GP1:91,2] = PR[GP1:90,2] + 33.290;
   1:L PR[91] 10mm/sec CNT100;
   1:  PR[GP1:91,1] = PR[GP1:90,1] + -37.057;
   1:  PR[GP1:91,2] = PR[GP1:90,2] + 34.580;
   1:L PR[91] 10mm/sec CNT100;
   1:  PR[GP1:91,1] = PR[GP1:90,1] + -41.465;
   1:  PR[GP1:91,2] = PR[GP1:90,2] + 34.219;
   1:L PR[91] 10mm/sec CNT100;
   1:  PR[GP1:91,1] = PR[GP1:90,1] + -47.899;
   1:  PR[GP1:91,2] = PR[GP1:90,2] + 33.242;
   1:L PR[91] 10mm/sec CNT100;
   1:  PR[GP1:91,1] = PR[GP1:90,1] + -53.288;
   1:  PR[GP1:91,2] = PR[GP1:90,2] + 30.899;
   1:L PR[91] 10mm/sec CNT100;
   1:  PR[GP1:91,1] = PR[GP1:90,1] + -57.932;
   1:  PR[GP1:91,2] = PR[GP1:90,2] + 28.580;
   1:L PR[91] 10mm/sec CNT100;
   1:  PR[GP1:91,1] = PR[GP1:90,1] + -63.071;
   1:  PR[GP1:91,2] = PR[GP1:90,2] + 23.893;
   1:L PR[91] 10mm/sec CNT100;
   1:  PR[GP1:91,1] = PR[GP1:90,1] + -66.064;
   1:  PR[GP1:91,2] = PR[GP1:90,2] + 20.947;
   1:L PR[91] 10mm/sec CNT100;
   1:  PR[GP1:91,1] = PR[GP1:90,1] + -69.728;
   1:  PR[GP1:91,2] = PR[GP1:90,2] + 14.236;
   1:L PR[91] 10mm/sec CNT100;
   1:  PR[GP1:91,1] = PR[GP1:90,1] + -71.364;
   1:  PR[GP1:91,2] = PR[GP1:90,2] + 11.072;
   1:L PR[91] 10mm/sec CNT100;
   1:  PR[GP1:91,1] = PR[GP1:90,1] + -72.728;
   1:  PR[GP1:91,2] = PR[GP1:90,2] + 3.014;
   1:L PR[91] 10mm/sec CNT100;
   1:  PR[GP1:91,1] = PR[GP1:90,1] + -73.211;
   1:  PR[GP1:91,2] = PR[GP1:90,2] + -0.002;
   1:L PR[91] 10mm/sec CNT100;
   1:  PR[GP1:91,1] = PR[GP1:90,1] + -71.879;
   1:  PR[GP1:91,2] = PR[GP1:90,2] + -7.854;
   1:L PR[91] 10mm/sec CNT100;
   1:  PR[GP1:91,1] = PR[GP1:90,1] + -71.362;
   1:  PR[GP1:91,2] = PR[GP1:90,2] + -11.083;
   1:L PR[91] 10mm/sec CNT100;
   1:  PR[GP1:91,1] = PR[GP1:90,1] + -69.728;
   1:  PR[GP1:91,2] = PR[GP1:90,2] + -14.245;
   1:L PR[91] 10mm/sec CNT100;
   1:  PR[GP1:91,1] = PR[GP1:90,1] + -66.064;
   1:  PR[GP1:91,2] = PR[GP1:90,2] + -20.956;
   1:L PR[91] 10mm/sec CNT100;
   1:  PR[GP1:91,1] = PR[GP1:90,1] + -63.071;
   1:  PR[GP1:91,2] = PR[GP1:90,2] + -23.902;
   1:L PR[91] 10mm/sec CNT100;
   1:  PR[GP1:91,1] = PR[GP1:90,1] + -57.932;
   1:  PR[GP1:91,2] = PR[GP1:90,2] + -28.589;
   1:L PR[91] 10mm/sec CNT100;
   1:  PR[GP1:91,1] = PR[GP1:90,1] + -53.288;
   1:  PR[GP1:91,2] = PR[GP1:90,2] + -30.908;
   1:L PR[91] 10mm/sec CNT100;
   1:  PR[GP1:91,1] = PR[GP1:90,1] + -47.899;
   1:  PR[GP1:91,2] = PR[GP1:90,2] + -33.251;
   1:L PR[91] 10mm/sec CNT100;
   1:  PR[GP1:91,1] = PR[GP1:90,1] + -41.465;
   1:  PR[GP1:91,2] = PR[GP1:90,2] + -34.228;
   1:L PR[91] 10mm/sec CNT100;
   1:  PR[GP1:91,1] = PR[GP1:90,1] + -37.057;
   1:  PR[GP1:91,2] = PR[GP1:90,2] + -34.589;
   1:L PR[91] 10mm/sec CNT100;
   1:  PR[GP1:91,1] = PR[GP1:90,1] + -29.094;
   1:  PR[GP1:91,2] = PR[GP1:90,2] + -33.298;
   1:L PR[91] 10mm/sec CNT100;
   1:  PR[GP1:91,1] = PR[GP1:90,1] + -26.487;
   1:  PR[GP1:91,2] = PR[GP1:90,2] + -32.643;
   1:L PR[91] 10mm/sec CNT100;
   1:  PR[GP1:91,1] = PR[GP1:90,1] + -17.844;
   1:  PR[GP1:91,2] = PR[GP1:90,2] + -28.224;
   1:L PR[91] 10mm/sec CNT100;
   1:  PR[GP1:91,1] = PR[GP1:90,1] + -17.120;
   1:  PR[GP1:91,2] = PR[GP1:90,2] + -27.753;
   1:L PR[91] 10mm/sec CNT100;
   1:  PR[GP1:91,1] = PR[GP1:90,1] + -12.636;
   1:  PR[GP1:91,2] = PR[GP1:90,2] + -23.257;
   1:L PR[91] 10mm/sec CNT100;
   1:  PR[GP1:91,1] = PR[GP1:90,1] + -9.604;
   1:  PR[GP1:91,2] = PR[GP1:90,2] + -20.329;
   1:L PR[91] 10mm/sec CNT100;
   1:  PR[GP1:91,1] = PR[GP1:90,1] + -9.275;
   1:  PR[GP1:91,2] = PR[GP1:90,2] + -19.852;
   1:L PR[91] 10mm/sec CNT100;
   1:  PR[GP1:91,1] = PR[GP1:90,1] + -4.689;
   1:  PR[GP1:91,2] = PR[GP1:90,2] + -11.079;
   1:L PR[91] 10mm/sec CNT100;
   1:  PR[GP1:91,1] = PR[GP1:90,1] + -4.456;
   1:  PR[GP1:91,2] = PR[GP1:90,2] + -10.403;
   1:L PR[91] 10mm/sec CNT100;
   1:  PR[GP1:91,1] = PR[GP1:90,1] + -3.875;
   1:  PR[GP1:91,2] = PR[GP1:90,2] + -9.761;
   1:L PR[91] 10mm/sec CNT100;
   1:  PR[GP1:91,1] = PR[GP1:90,1] + -3.742;
   1:  PR[GP1:91,2] = PR[GP1:90,2] + -9.679;
   1:L PR[91] 10mm/sec CNT100;
   1:  PR[GP1:91,1] = PR[GP1:90,1] + -1.610;
   1:  PR[GP1:91,2] = PR[GP1:90,2] + -7.132;
   1:L PR[91] 10mm/sec CNT100;
   1:  PR[GP1:91,1] = PR[GP1:90,1] + 0.379;
   1:  PR[GP1:91,2] = PR[GP1:90,2] + -7.285;
   1:L PR[91] 10mm/sec CNT100;
   1:  PR[GP1:91,1] = PR[GP1:90,1] + 0.448;
   1:  PR[GP1:91,2] = PR[GP1:90,2] + -7.341;
   1:L PR[91] 10mm/sec CNT100;
   1:  PR[GP1:91,1] = PR[GP1:90,1] + 2.794;
   1:  PR[GP1:91,2] = PR[GP1:90,2] + -7.317;
   1:L PR[91] 10mm/sec CNT100;
   1:  PR[GP1:91,1] = PR[GP1:90,1] + 3.638;
   1:  PR[GP1:91,2] = PR[GP1:90,2] + -8.922;
   1:L PR[91] 10mm/sec CNT100;
   1:  PR[GP1:91,1] = PR[GP1:90,1] + 4.759;
   1:  PR[GP1:91,2] = PR[GP1:90,2] + -10.213;
   1:L PR[91] 10mm/sec CNT100;
   1:  PR[GP1:91,1] = PR[GP1:90,1] + 5.446;
   1:  PR[GP1:91,2] = PR[GP1:90,2] + -10.966;
   1:L PR[91] 10mm/sec CNT100;
   1:  PR[GP1:91,1] = PR[GP1:90,1] + 10.085;
   1:  PR[GP1:91,2] = PR[GP1:90,2] + -19.826;
   1:L PR[91] 10mm/sec CNT100;
   1:  PR[GP1:91,1] = PR[GP1:90,1] + 10.415;
   1:  PR[GP1:91,2] = PR[GP1:90,2] + -20.306;
   1:L PR[91] 10mm/sec CNT100;
   1:  PR[GP1:91,1] = PR[GP1:90,1] + 13.457;
   1:  PR[GP1:91,2] = PR[GP1:90,2] + -23.251;
   1:L PR[91] 10mm/sec CNT100;
   1:  PR[GP1:91,1] = PR[GP1:90,1] + 17.929;
   1:  PR[GP1:91,2] = PR[GP1:90,2] + -27.748;
   1:L PR[91] 10mm/sec CNT100;
   1:  PR[GP1:91,1] = PR[GP1:90,1] + 18.652;
   1:  PR[GP1:91,2] = PR[GP1:90,2] + -28.217;
   1:L PR[91] 10mm/sec CNT100;
   1:  PR[GP1:91,1] = PR[GP1:90,1] + 27.297;
   1:  PR[GP1:91,2] = PR[GP1:90,2] + -32.638;
   1:L PR[91] 10mm/sec CNT100;
   1:  PR[GP1:91,1] = PR[GP1:90,1] + 29.903;
   1:  PR[GP1:91,2] = PR[GP1:90,2] + -33.293;
   1:L PR[91] 10mm/sec CNT100;
   1:  PR[GP1:91,1] = PR[GP1:90,1] + 37.870;
   1:  PR[GP1:91,2] = PR[GP1:90,2] + -34.589;
   1:L PR[91] 10mm/sec CNT100;
   1:  PR[GP1:91,1] = PR[GP1:90,1] + 42.277;
   1:  PR[GP1:91,2] = PR[GP1:90,2] + -34.228;
   1:L PR[91] 10mm/sec CNT100;
   1:  PR[GP1:91,1] = PR[GP1:90,1] + 48.714;
   1:  PR[GP1:91,2] = PR[GP1:90,2] + -33.251;
   1:L PR[91] 10mm/sec CNT100;
   1:  PR[GP1:91,1] = PR[GP1:90,1] + 54.104;
   1:  PR[GP1:91,2] = PR[GP1:90,2] + -30.909;
   1:L PR[91] 10mm/sec CNT100;
   1:  PR[GP1:91,1] = PR[GP1:90,1] + 58.749;
   1:  PR[GP1:91,2] = PR[GP1:90,2] + -28.593;
   1:L PR[91] 10mm/sec CNT100;
   1:  PR[GP1:91,1] = PR[GP1:90,1] + 63.888;
   1:  PR[GP1:91,2] = PR[GP1:90,2] + -23.904;
   1:L PR[91] 10mm/sec CNT100;
   1:  PR[GP1:91,1] = PR[GP1:90,1] + 66.884;
   1:  PR[GP1:91,2] = PR[GP1:90,2] + -20.953;
   1:L PR[91] 10mm/sec CNT100;
   1:  PR[GP1:91,1] = PR[GP1:90,1] + 70.548;
   1:  PR[GP1:91,2] = PR[GP1:90,2] + -14.246;
   1:L PR[91] 10mm/sec CNT100;
   1:  PR[GP1:91,1] = PR[GP1:90,1] + 72.184;
   1:  PR[GP1:91,2] = PR[GP1:90,2] + -11.090;
   1:L PR[91] 10mm/sec CNT100;
   1:  PR[GP1:91,1] = PR[GP1:90,1] + 73.548;
   1:  PR[GP1:91,2] = PR[GP1:90,2] + -3.028;
   1:L PR[91] 10mm/sec CNT100;
   1:  PR[GP1:91,1] = PR[GP1:90,1] + 74.032;
   1:  PR[GP1:91,2] = PR[GP1:90,2] + -0.007;
   1:L PR[91] 10mm/sec CNT100;
   1:  PR[GP1:91,1] = PR[GP1:90,1] + 72.700;
   1:  PR[GP1:91,2] = PR[GP1:90,2] + 7.849;
   1:L PR[91] 10mm/sec CNT100;
   1:  PR[GP1:91,1] = PR[GP1:90,1] + 72.183;
   1:  PR[GP1:91,2] = PR[GP1:90,2] + 11.083;
   1:L PR[91] 10mm/sec CNT100;
   1:  PR[GP1:91,1] = PR[GP1:90,1] + 70.548;
   1:  PR[GP1:91,2] = PR[GP1:90,2] + 14.238;
   1:L PR[91] 10mm/sec CNT100;
   1:  PR[GP1:91,1] = PR[GP1:90,1] + 66.883;
   1:  PR[GP1:91,2] = PR[GP1:90,2] + 20.944;
   1:L PR[91] 10mm/sec CNT100;
   1:  PR[GP1:91,1] = PR[GP1:90,1] + 63.888;
   1:  PR[GP1:91,2] = PR[GP1:90,2] + 23.895;
   1:L PR[91] 10mm/sec CNT100;
   1:  PR[GP1:91,1] = PR[GP1:90,1] + 58.749;
   1:  PR[GP1:91,2] = PR[GP1:90,2] + 28.584;
   1:L PR[91] 10mm/sec CNT100;
   1:  PR[GP1:91,1] = PR[GP1:90,1] + 54.104;
   1:  PR[GP1:91,2] = PR[GP1:90,2] + 30.900;
   1:L PR[91] 10mm/sec CNT100;
   1:  PR[GP1:91,1] = PR[GP1:90,1] + 48.714;
   1:  PR[GP1:91,2] = PR[GP1:90,2] + 33.242;
   1:L PR[91] 10mm/sec CNT100;
   1:  PR[GP1:91,1] = PR[GP1:90,1] + 42.277;
   1:  PR[GP1:91,2] = PR[GP1:90,2] + 34.219;
   1:L PR[91] 10mm/sec CNT100;
   1:  PR[GP1:91,1] = PR[GP1:90,1] + 37.870;
   1:  PR[GP1:91,2] = PR[GP1:90,2] + 34.581;
   1:L PR[91] 10mm/sec CNT100;
   1:  PR[GP1:91,1] = PR[GP1:90,1] + 29.903;
   1:  PR[GP1:91,2] = PR[GP1:90,2] + 33.284;
   1:L PR[91] 10mm/sec CNT100;
   1:  PR[GP1:91,1] = PR[GP1:90,1] + 27.297;
   1:  PR[GP1:91,2] = PR[GP1:90,2] + 32.629;
   1:L PR[91] 10mm/sec CNT100;
   1:  PR[GP1:91,1] = PR[GP1:90,1] + 18.651;
   1:  PR[GP1:91,2] = PR[GP1:90,2] + 28.208;
   1:L PR[91] 10mm/sec CNT100;
   1:  PR[GP1:91,1] = PR[GP1:90,1] + 17.929;
   1:  PR[GP1:91,2] = PR[GP1:90,2] + 27.739;
   1:L PR[91] 10mm/sec CNT100;
   1:  PR[GP1:91,1] = PR[GP1:90,1] + 13.457;
   1:  PR[GP1:91,2] = PR[GP1:90,2] + 23.242;
   1:L PR[91] 10mm/sec CNT100;
   1:  PR[GP1:91,1] = PR[GP1:90,1] + 10.415;
   1:  PR[GP1:91,2] = PR[GP1:90,2] + 20.297;
   1:L PR[91] 10mm/sec CNT100;
   1:  PR[GP1:91,1] = PR[GP1:90,1] + 10.086;
   1:  PR[GP1:91,2] = PR[GP1:90,2] + 19.820;
   1:L PR[91] 10mm/sec CNT100;
   1:  PR[GP1:91,1] = PR[GP1:90,1] + 5.503;
   1:  PR[GP1:91,2] = PR[GP1:90,2] + 11.066;
   1:L PR[91] 10mm/sec CNT100;
   1:  PR[GP1:91,1] = PR[GP1:90,1] + 5.268;
   1:  PR[GP1:91,2] = PR[GP1:90,2] + 10.382;
   1:L PR[91] 10mm/sec CNT100;
   1:  PR[GP1:91,1] = PR[GP1:90,1] + 3.384;
   1:  PR[GP1:91,2] = PR[GP1:90,2] + 8.100;
   1:L PR[91] 10mm/sec CNT100;
   1:  PR[GP1:91,1] = PR[GP1:90,1] + 2.704;
   1:  PR[GP1:91,2] = PR[GP1:90,2] + 7.360;
   1:L PR[91] 10mm/sec CNT100;
   1:  PR[GP1:91,1] = PR[GP1:90,1] + 2.272;
   1:  PR[GP1:91,2] = PR[GP1:90,2] + 7.121;
   1:L PR[91] 10mm/sec CNT100;
   1:  PR[GP1:91,1] = PR[GP1:90,1] + -0.539;
   1:  PR[GP1:91,2] = PR[GP1:90,2] + 8.308;
   1:  PR[GP1:91,3] = PR[GP1:90,3] + 25.270;
   1:L PR[91] 10mm/sec CNT100;
   1:  PR[GP1:91,1] = PR[GP1:90,1] + -1.715;
   1:  PR[GP1:91,2] = PR[GP1:90,2] + 8.397;
   1:L PR[91] 10mm/sec CNT100;
   1:  PR[GP1:91,1] = PR[GP1:90,1] + -1.987;
   1:  PR[GP1:91,2] = PR[GP1:90,2] + 8.588;
   1:L PR[91] 10mm/sec CNT100;
   1:  PR[GP1:91,1] = PR[GP1:90,1] + -4.361;
   1:  PR[GP1:91,2] = PR[GP1:90,2] + 11.497;
   1:L PR[91] 10mm/sec CNT100;
   1:  PR[GP1:91,1] = PR[GP1:90,1] + -4.598;
   1:  PR[GP1:91,2] = PR[GP1:90,2] + 11.923;
   1:L PR[91] 10mm/sec CNT100;
   1:  PR[GP1:91,1] = PR[GP1:90,1] + -8.162;
   1:  PR[GP1:91,2] = PR[GP1:90,2] + 18.729;
   1:L PR[91] 10mm/sec CNT100;
   1:  PR[GP1:91,1] = PR[GP1:90,1] + -9.700;
   1:  PR[GP1:91,2] = PR[GP1:90,2] + 20.957;
   1:L PR[91] 10mm/sec CNT100;
   1:  PR[GP1:91,1] = PR[GP1:90,1] + -16.516;
   1:  PR[GP1:91,2] = PR[GP1:90,2] + 27.540;
   1:L PR[91] 10mm/sec CNT100;
   1:  PR[GP1:91,1] = PR[GP1:90,1] + -17.274;
   1:  PR[GP1:91,2] = PR[GP1:90,2] + 28.125;
   1:L PR[91] 10mm/sec CNT100;
   1:  PR[GP1:91,1] = PR[GP1:90,1] + -22.301;
   1:  PR[GP1:91,2] = PR[GP1:90,2] + 30.577;
   1:L PR[91] 10mm/sec CNT100;
   1:  PR[GP1:91,1] = PR[GP1:90,1] + -26.768;
   1:  PR[GP1:91,2] = PR[GP1:90,2] + 32.861;
   1:L PR[91] 10mm/sec CNT100;
   1:  PR[GP1:91,1] = PR[GP1:90,1] + -27.546;
   1:  PR[GP1:91,2] = PR[GP1:90,2] + 33.057;
   1:L PR[91] 10mm/sec CNT100;
   1:  PR[GP1:91,1] = PR[GP1:90,1] + -37.274;
   1:  PR[GP1:91,2] = PR[GP1:90,2] + 34.634;
   1:L PR[91] 10mm/sec CNT100;
   1:  PR[GP1:91,1] = PR[GP1:90,1] + -39.942;
   1:  PR[GP1:91,2] = PR[GP1:90,2] + 34.415;
   1:L PR[91] 10mm/sec CNT100;
   1:  PR[GP1:91,1] = PR[GP1:90,1] + -48.019;
   1:  PR[GP1:91,2] = PR[GP1:90,2] + 33.188;
   1:L PR[91] 10mm/sec CNT100;
   1:  PR[GP1:91,1] = PR[GP1:90,1] + -51.929;
   1:  PR[GP1:91,2] = PR[GP1:90,2] + 31.488;
   1:L PR[91] 10mm/sec CNT100;
   1:  PR[GP1:91,1] = PR[GP1:90,1] + -57.950;
   1:  PR[GP1:91,2] = PR[GP1:90,2] + 28.481;
   1:L PR[91] 10mm/sec CNT100;
   1:  PR[GP1:91,1] = PR[GP1:90,1] + -61.982;
   1:  PR[GP1:91,2] = PR[GP1:90,2] + 24.804;
   1:L PR[91] 10mm/sec CNT100;
   1:  PR[GP1:91,1] = PR[GP1:90,1] + -65.997;
   1:  PR[GP1:91,2] = PR[GP1:90,2] + 20.853;
   1:L PR[91] 10mm/sec CNT100;
   1:  PR[GP1:91,1] = PR[GP1:90,1] + -68.987;
   1:  PR[GP1:91,2] = PR[GP1:90,2] + 15.377;
   1:L PR[91] 10mm/sec CNT100;
   1:  PR[GP1:91,1] = PR[GP1:90,1] + -71.240;
   1:  PR[GP1:91,2] = PR[GP1:90,2] + 11.017;
   1:L PR[91] 10mm/sec CNT100;
   1:  PR[GP1:91,1] = PR[GP1:90,1] + -72.374;
   1:  PR[GP1:91,2] = PR[GP1:90,2] + 4.314;
   1:L PR[91] 10mm/sec CNT100;
   1:  PR[GP1:91,1] = PR[GP1:90,1] + -73.066;
   1:  PR[GP1:91,2] = PR[GP1:90,2] + -0.002;
   1:L PR[91] 10mm/sec CNT100;
   1:  PR[GP1:91,1] = PR[GP1:90,1] + -71.951;
   1:  PR[GP1:91,2] = PR[GP1:90,2] + -6.579;
   1:L PR[91] 10mm/sec CNT100;
   1:  PR[GP1:91,1] = PR[GP1:90,1] + -71.239;
   1:  PR[GP1:91,2] = PR[GP1:90,2] + -11.028;
   1:L PR[91] 10mm/sec CNT100;
   1:  PR[GP1:91,1] = PR[GP1:90,1] + -68.987;
   1:  PR[GP1:91,2] = PR[GP1:90,2] + -15.385;
   1:L PR[91] 10mm/sec CNT100;
   1:  PR[GP1:91,1] = PR[GP1:90,1] + -65.997;
   1:  PR[GP1:91,2] = PR[GP1:90,2] + -20.861;
   1:L PR[91] 10mm/sec CNT100;
   1:  PR[GP1:91,1] = PR[GP1:90,1] + -61.982;
   1:  PR[GP1:91,2] = PR[GP1:90,2] + -24.812;
   1:L PR[91] 10mm/sec CNT100;
   1:  PR[GP1:91,1] = PR[GP1:90,1] + -57.950;
   1:  PR[GP1:91,2] = PR[GP1:90,2] + -28.490;
   1:L PR[91] 10mm/sec CNT100;
   1:  PR[GP1:91,1] = PR[GP1:90,1] + -51.929;
   1:  PR[GP1:91,2] = PR[GP1:90,2] + -31.497;
   1:L PR[91] 10mm/sec CNT100;
   1:  PR[GP1:91,1] = PR[GP1:90,1] + -48.019;
   1:  PR[GP1:91,2] = PR[GP1:90,2] + -33.197;
   1:L PR[91] 10mm/sec CNT100;
   1:  PR[GP1:91,1] = PR[GP1:90,1] + -39.942;
   1:  PR[GP1:91,2] = PR[GP1:90,2] + -34.424;
   1:L PR[91] 10mm/sec CNT100;
   1:  PR[GP1:91,1] = PR[GP1:90,1] + -37.274;
   1:  PR[GP1:91,2] = PR[GP1:90,2] + -34.642;
   1:L PR[91] 10mm/sec CNT100;
   1:  PR[GP1:91,1] = PR[GP1:90,1] + -27.546;
   1:  PR[GP1:91,2] = PR[GP1:90,2] + -33.065;
   1:L PR[91] 10mm/sec CNT100;
   1:  PR[GP1:91,1] = PR[GP1:90,1] + -26.768;
   1:  PR[GP1:91,2] = PR[GP1:90,2] + -32.870;
   1:L PR[91] 10mm/sec CNT100;
   1:  PR[GP1:91,1] = PR[GP1:90,1] + -22.301;
   1:  PR[GP1:91,2] = PR[GP1:90,2] + -30.585;
   1:L PR[91] 10mm/sec CNT100;
   1:  PR[GP1:91,1] = PR[GP1:90,1] + -17.274;
   1:  PR[GP1:91,2] = PR[GP1:90,2] + -28.134;
   1:L PR[91] 10mm/sec CNT100;
   1:  PR[GP1:91,1] = PR[GP1:90,1] + -16.516;
   1:  PR[GP1:91,2] = PR[GP1:90,2] + -27.549;
   1:L PR[91] 10mm/sec CNT100;
   1:  PR[GP1:91,1] = PR[GP1:90,1] + -9.700;
   1:  PR[GP1:91,2] = PR[GP1:90,2] + -20.966;
   1:L PR[91] 10mm/sec CNT100;
   1:  PR[GP1:91,1] = PR[GP1:90,1] + -8.156;
   1:  PR[GP1:91,2] = PR[GP1:90,2] + -18.727;
   1:L PR[91] 10mm/sec CNT100;
   1:  PR[GP1:91,1] = PR[GP1:90,1] + -4.605;
   1:  PR[GP1:91,2] = PR[GP1:90,2] + -11.930;
   1:L PR[91] 10mm/sec CNT100;
   1:  PR[GP1:91,1] = PR[GP1:90,1] + -4.530;
   1:  PR[GP1:91,2] = PR[GP1:90,2] + -11.712;
   1:L PR[91] 10mm/sec CNT100;
   1:  PR[GP1:91,1] = PR[GP1:90,1] + -4.439;
   1:  PR[GP1:91,2] = PR[GP1:90,2] + -11.611;
   1:L PR[91] 10mm/sec CNT100;
   1:  PR[GP1:91,1] = PR[GP1:90,1] + -4.362;
   1:  PR[GP1:91,2] = PR[GP1:90,2] + -11.463;
   1:L PR[91] 10mm/sec CNT100;
   1:  PR[GP1:91,1] = PR[GP1:90,1] + -4.318;
   1:  PR[GP1:91,2] = PR[GP1:90,2] + -11.478;
   1:L PR[91] 10mm/sec CNT100;
   1:  PR[GP1:91,1] = PR[GP1:90,1] + -4.248;
   1:  PR[GP1:91,2] = PR[GP1:90,2] + -11.400;
   1:L PR[91] 10mm/sec CNT100;
   1:  PR[GP1:91,1] = PR[GP1:90,1] + -4.212;
   1:  PR[GP1:91,2] = PR[GP1:90,2] + -11.378;
   1:L PR[91] 10mm/sec CNT100;
   1:  PR[GP1:91,1] = PR[GP1:90,1] + -1.631;
   1:  PR[GP1:91,2] = PR[GP1:90,2] + -8.295;
   1:L PR[91] 10mm/sec CNT100;
   1:  PR[GP1:91,1] = PR[GP1:90,1] + -0.160;
   1:  PR[GP1:91,2] = PR[GP1:90,2] + -8.408;
   1:L PR[91] 10mm/sec CNT100;
   1:  PR[GP1:91,1] = PR[GP1:90,1] + -0.122;
   1:  PR[GP1:91,2] = PR[GP1:90,2] + -8.438;
   1:L PR[91] 10mm/sec CNT100;
   1:  PR[GP1:91,1] = PR[GP1:90,1] + 2.697;
   1:  PR[GP1:91,2] = PR[GP1:90,2] + -8.409;
   1:L PR[91] 10mm/sec CNT100;
   1:  PR[GP1:91,1] = PR[GP1:90,1] + 3.297;
   1:  PR[GP1:91,2] = PR[GP1:90,2] + -9.552;
   1:L PR[91] 10mm/sec CNT100;
   1:  PR[GP1:91,1] = PR[GP1:90,1] + 4.014;
   1:  PR[GP1:91,2] = PR[GP1:90,2] + -10.378;
   1:L PR[91] 10mm/sec CNT100;
   1:  PR[GP1:91,1] = PR[GP1:90,1] + 5.378;
   1:  PR[GP1:91,2] = PR[GP1:90,2] + -11.864;
   1:L PR[91] 10mm/sec CNT100;
   1:  PR[GP1:91,1] = PR[GP1:90,1] + 8.966;
   1:  PR[GP1:91,2] = PR[GP1:90,2] + -18.703;
   1:L PR[91] 10mm/sec CNT100;
   1:  PR[GP1:91,1] = PR[GP1:90,1] + 10.513;
   1:  PR[GP1:91,2] = PR[GP1:90,2] + -20.946;
   1:L PR[91] 10mm/sec CNT100;
   1:  PR[GP1:91,1] = PR[GP1:90,1] + 17.324;
   1:  PR[GP1:91,2] = PR[GP1:90,2] + -27.542;
   1:L PR[91] 10mm/sec CNT100;
   1:  PR[GP1:91,1] = PR[GP1:90,1] + 18.083;
   1:  PR[GP1:91,2] = PR[GP1:90,2] + -28.129;
   1:L PR[91] 10mm/sec CNT100;
   1:  PR[GP1:91,1] = PR[GP1:90,1] + 23.121;
   1:  PR[GP1:91,2] = PR[GP1:90,2] + -30.586;
   1:L PR[91] 10mm/sec CNT100;
   1:  PR[GP1:91,1] = PR[GP1:90,1] + 27.577;
   1:  PR[GP1:91,2] = PR[GP1:90,2] + -32.864;
   1:L PR[91] 10mm/sec CNT100;
   1:  PR[GP1:91,1] = PR[GP1:90,1] + 28.353;
   1:  PR[GP1:91,2] = PR[GP1:90,2] + -33.059;
   1:L PR[91] 10mm/sec CNT100;
   1:  PR[GP1:91,1] = PR[GP1:90,1] + 38.086;
   1:  PR[GP1:91,2] = PR[GP1:90,2] + -34.643;
   1:L PR[91] 10mm/sec CNT100;
   1:  PR[GP1:91,1] = PR[GP1:90,1] + 40.753;
   1:  PR[GP1:91,2] = PR[GP1:90,2] + -34.424;
   1:L PR[91] 10mm/sec CNT100;
   1:  PR[GP1:91,1] = PR[GP1:90,1] + 48.833;
   1:  PR[GP1:91,2] = PR[GP1:90,2] + -33.197;
   1:L PR[91] 10mm/sec CNT100;
   1:  PR[GP1:91,1] = PR[GP1:90,1] + 52.743;
   1:  PR[GP1:91,2] = PR[GP1:90,2] + -31.498;
   1:L PR[91] 10mm/sec CNT100;
   1:  PR[GP1:91,1] = PR[GP1:90,1] + 58.767;
   1:  PR[GP1:91,2] = PR[GP1:90,2] + -28.495;
   1:L PR[91] 10mm/sec CNT100;
   1:  PR[GP1:91,1] = PR[GP1:90,1] + 62.799;
   1:  PR[GP1:91,2] = PR[GP1:90,2] + -24.816;
   1:L PR[91] 10mm/sec CNT100;
   1:  PR[GP1:91,1] = PR[GP1:90,1] + 66.816;
   1:  PR[GP1:91,2] = PR[GP1:90,2] + -20.858;
   1:L PR[91] 10mm/sec CNT100;
   1:  PR[GP1:91,1] = PR[GP1:90,1] + 69.806;
   1:  PR[GP1:91,2] = PR[GP1:90,2] + -15.385;
   1:L PR[91] 10mm/sec CNT100;
   1:  PR[GP1:91,1] = PR[GP1:90,1] + 72.060;
   1:  PR[GP1:91,2] = PR[GP1:90,2] + -11.036;
   1:L PR[91] 10mm/sec CNT100;
   1:  PR[GP1:91,1] = PR[GP1:90,1] + 73.195;
   1:  PR[GP1:91,2] = PR[GP1:90,2] + -4.330;
   1:L PR[91] 10mm/sec CNT100;
   1:  PR[GP1:91,1] = PR[GP1:90,1] + 73.887;
   1:  PR[GP1:91,2] = PR[GP1:90,2] + -0.007;
   1:L PR[91] 10mm/sec CNT100;
   1:  PR[GP1:91,1] = PR[GP1:90,1] + 72.771;
   1:  PR[GP1:91,2] = PR[GP1:90,2] + 6.573;
   1:L PR[91] 10mm/sec CNT100;
   1:  PR[GP1:91,1] = PR[GP1:90,1] + 72.059;
   1:  PR[GP1:91,2] = PR[GP1:90,2] + 11.030;
   1:L PR[91] 10mm/sec CNT100;
   1:  PR[GP1:91,1] = PR[GP1:90,1] + 69.806;
   1:  PR[GP1:91,2] = PR[GP1:90,2] + 15.377;
   1:L PR[91] 10mm/sec CNT100;
   1:  PR[GP1:91,1] = PR[GP1:90,1] + 66.816;
   1:  PR[GP1:91,2] = PR[GP1:90,2] + 20.849;
   1:L PR[91] 10mm/sec CNT100;
   1:  PR[GP1:91,1] = PR[GP1:90,1] + 62.799;
   1:  PR[GP1:91,2] = PR[GP1:90,2] + 24.807;
   1:L PR[91] 10mm/sec CNT100;
   1:  PR[GP1:91,1] = PR[GP1:90,1] + 58.767;
   1:  PR[GP1:91,2] = PR[GP1:90,2] + 28.486;
   1:L PR[91] 10mm/sec CNT100;
   1:  PR[GP1:91,1] = PR[GP1:90,1] + 52.743;
   1:  PR[GP1:91,2] = PR[GP1:90,2] + 31.490;
   1:L PR[91] 10mm/sec CNT100;
   1:  PR[GP1:91,1] = PR[GP1:90,1] + 48.833;
   1:  PR[GP1:91,2] = PR[GP1:90,2] + 33.188;
   1:L PR[91] 10mm/sec CNT100;
   1:  PR[GP1:91,1] = PR[GP1:90,1] + 40.752;
   1:  PR[GP1:91,2] = PR[GP1:90,2] + 34.415;
   1:L PR[91] 10mm/sec CNT100;
   1:  PR[GP1:91,1] = PR[GP1:90,1] + 38.086;
   1:  PR[GP1:91,2] = PR[GP1:90,2] + 34.634;
   1:L PR[91] 10mm/sec CNT100;
   1:  PR[GP1:91,1] = PR[GP1:90,1] + 28.353;
   1:  PR[GP1:91,2] = PR[GP1:90,2] + 33.050;
   1:L PR[91] 10mm/sec CNT100;
   1:  PR[GP1:91,1] = PR[GP1:90,1] + 27.577;
   1:  PR[GP1:91,2] = PR[GP1:90,2] + 32.855;
   1:L PR[91] 10mm/sec CNT100;
   1:  PR[GP1:91,1] = PR[GP1:90,1] + 23.121;
   1:  PR[GP1:91,2] = PR[GP1:90,2] + 30.577;
   1:L PR[91] 10mm/sec CNT100;
   1:  PR[GP1:91,1] = PR[GP1:90,1] + 18.083;
   1:  PR[GP1:91,2] = PR[GP1:90,2] + 28.120;
   1:L PR[91] 10mm/sec CNT100;
   1:  PR[GP1:91,1] = PR[GP1:90,1] + 17.324;
   1:  PR[GP1:91,2] = PR[GP1:90,2] + 27.533;
   1:L PR[91] 10mm/sec CNT100;
   1:  PR[GP1:91,1] = PR[GP1:90,1] + 10.513;
   1:  PR[GP1:91,2] = PR[GP1:90,2] + 20.937;
   1:L PR[91] 10mm/sec CNT100;
   1:  PR[GP1:91,1] = PR[GP1:90,1] + 8.972;
   1:  PR[GP1:91,2] = PR[GP1:90,2] + 18.706;
   1:L PR[91] 10mm/sec CNT100;
   1:  PR[GP1:91,1] = PR[GP1:90,1] + 5.435;
   1:  PR[GP1:91,2] = PR[GP1:90,2] + 11.964;
   1:L PR[91] 10mm/sec CNT100;
   1:  PR[GP1:91,1] = PR[GP1:90,1] + 5.340;
   1:  PR[GP1:91,2] = PR[GP1:90,2] + 11.686;
   1:L PR[91] 10mm/sec CNT100;
   1:  PR[GP1:91,1] = PR[GP1:90,1] + 3.115;
   1:  PR[GP1:91,2] = PR[GP1:90,2] + 8.991;
   1:L PR[91] 10mm/sec CNT100;
   1:  PR[GP1:91,1] = PR[GP1:90,1] + 2.643;
   1:  PR[GP1:91,2] = PR[GP1:90,2] + 8.478;
   1:L PR[91] 10mm/sec CNT100;
   1:  PR[GP1:91,1] = PR[GP1:90,1] + 2.283;
   1:  PR[GP1:91,2] = PR[GP1:90,2] + 8.278;
   1:L PR[91] 10mm/sec CNT100;
   1:  PR[GP1:91,1] = PR[GP1:90,1] + -1.013;
   1:  PR[GP1:91,2] = PR[GP1:90,2] + 9.470;
   1:  PR[GP1:91,3] = PR[GP1:90,3] + 26.600;
   1:L PR[91] 10mm/sec CNT100;
   1:  PR[GP1:91,1] = PR[GP1:90,1] + -1.664;
   1:  PR[GP1:91,2] = PR[GP1:90,2] + 9.520;
   1:L PR[91] 10mm/sec CNT100;
   1:  PR[GP1:91,1] = PR[GP1:90,1] + -1.900;
   1:  PR[GP1:91,2] = PR[GP1:90,2] + 9.685;
   1:L PR[91] 10mm/sec CNT100;
   1:  PR[GP1:91,1] = PR[GP1:90,1] + -3.590;
   1:  PR[GP1:91,2] = PR[GP1:90,2] + 11.756;
   1:L PR[91] 10mm/sec CNT100;
   1:  PR[GP1:91,1] = PR[GP1:90,1] + -4.493;
   1:  PR[GP1:91,2] = PR[GP1:90,2] + 12.731;
   1:L PR[91] 10mm/sec CNT100;
   1:  PR[GP1:91,1] = PR[GP1:90,1] + -7.048;
   1:  PR[GP1:91,2] = PR[GP1:90,2] + 17.613;
   1:L PR[91] 10mm/sec CNT100;
   1:  PR[GP1:91,1] = PR[GP1:90,1] + -9.796;
   1:  PR[GP1:91,2] = PR[GP1:90,2] + 21.594;
   1:L PR[91] 10mm/sec CNT100;
   1:  PR[GP1:91,1] = PR[GP1:90,1] + -15.094;
   1:  PR[GP1:91,2] = PR[GP1:90,2] + 26.710;
   1:L PR[91] 10mm/sec CNT100;
   1:  PR[GP1:91,1] = PR[GP1:90,1] + -17.434;
   1:  PR[GP1:91,2] = PR[GP1:90,2] + 28.517;
   1:L PR[91] 10mm/sec CNT100;
   1:  PR[GP1:91,1] = PR[GP1:90,1] + -26.057;
   1:  PR[GP1:91,2] = PR[GP1:90,2] + 32.723;
   1:L PR[91] 10mm/sec CNT100;
   1:  PR[GP1:91,1] = PR[GP1:90,1] + -26.916;
   1:  PR[GP1:91,2] = PR[GP1:90,2] + 33.050;
   1:L PR[91] 10mm/sec CNT100;
   1:  PR[GP1:91,1] = PR[GP1:90,1] + -31.930;
   1:  PR[GP1:91,2] = PR[GP1:90,2] + 33.785;
   1:L PR[91] 10mm/sec CNT100;
   1:  PR[GP1:91,1] = PR[GP1:90,1] + -37.491;
   1:  PR[GP1:91,2] = PR[GP1:90,2] + 34.687;
   1:L PR[91] 10mm/sec CNT100;
   1:  PR[GP1:91,1] = PR[GP1:90,1] + -38.419;
   1:  PR[GP1:91,2] = PR[GP1:90,2] + 34.611;
   1:L PR[91] 10mm/sec CNT100;
   1:  PR[GP1:91,1] = PR[GP1:90,1] + -48.138;
   1:  PR[GP1:91,2] = PR[GP1:90,2] + 33.134;
   1:L PR[91] 10mm/sec CNT100;
   1:  PR[GP1:91,1] = PR[GP1:90,1] + -50.569;
   1:  PR[GP1:91,2] = PR[GP1:90,2] + 32.078;
   1:L PR[91] 10mm/sec CNT100;
   1:  PR[GP1:91,1] = PR[GP1:90,1] + -57.968;
   1:  PR[GP1:91,2] = PR[GP1:90,2] + 28.383;
   1:L PR[91] 10mm/sec CNT100;
   1:  PR[GP1:91,1] = PR[GP1:90,1] + -60.894;
   1:  PR[GP1:91,2] = PR[GP1:90,2] + 25.714;
   1:L PR[91] 10mm/sec CNT100;
   1:  PR[GP1:91,1] = PR[GP1:90,1] + -65.929;
   1:  PR[GP1:91,2] = PR[GP1:90,2] + 20.758;
   1:L PR[91] 10mm/sec CNT100;
   1:  PR[GP1:91,1] = PR[GP1:90,1] + -68.245;
   1:  PR[GP1:91,2] = PR[GP1:90,2] + 16.517;
   1:L PR[91] 10mm/sec CNT100;
   1:  PR[GP1:91,1] = PR[GP1:90,1] + -71.116;
   1:  PR[GP1:91,2] = PR[GP1:90,2] + 10.962;
   1:L PR[91] 10mm/sec CNT100;
   1:  PR[GP1:91,1] = PR[GP1:90,1] + -72.021;
   1:  PR[GP1:91,2] = PR[GP1:90,2] + 5.614;
   1:L PR[91] 10mm/sec CNT100;
   1:  PR[GP1:91,1] = PR[GP1:90,1] + -72.921;
   1:  PR[GP1:91,2] = PR[GP1:90,2] + -0.002;
   1:L PR[91] 10mm/sec CNT100;
   1:  PR[GP1:91,1] = PR[GP1:90,1] + -72.022;
   1:  PR[GP1:91,2] = PR[GP1:90,2] + -5.303;
   1:L PR[91] 10mm/sec CNT100;
   1:  PR[GP1:91,1] = PR[GP1:90,1] + -71.115;
   1:  PR[GP1:91,2] = PR[GP1:90,2] + -10.973;
   1:L PR[91] 10mm/sec CNT100;
   1:  PR[GP1:91,1] = PR[GP1:90,1] + -68.245;
   1:  PR[GP1:91,2] = PR[GP1:90,2] + -16.526;
   1:L PR[91] 10mm/sec CNT100;
   1:  PR[GP1:91,1] = PR[GP1:90,1] + -65.929;
   1:  PR[GP1:91,2] = PR[GP1:90,2] + -20.767;
   1:L PR[91] 10mm/sec CNT100;
   1:  PR[GP1:91,1] = PR[GP1:90,1] + -60.893;
   1:  PR[GP1:91,2] = PR[GP1:90,2] + -25.723;
   1:L PR[91] 10mm/sec CNT100;
   1:  PR[GP1:91,1] = PR[GP1:90,1] + -57.968;
   1:  PR[GP1:91,2] = PR[GP1:90,2] + -28.392;
   1:L PR[91] 10mm/sec CNT100;
   1:  PR[GP1:91,1] = PR[GP1:90,1] + -50.569;
   1:  PR[GP1:91,2] = PR[GP1:90,2] + -32.086;
   1:L PR[91] 10mm/sec CNT100;
   1:  PR[GP1:91,1] = PR[GP1:90,1] + -48.139;
   1:  PR[GP1:91,2] = PR[GP1:90,2] + -33.143;
   1:L PR[91] 10mm/sec CNT100;
   1:  PR[GP1:91,1] = PR[GP1:90,1] + -38.420;
   1:  PR[GP1:91,2] = PR[GP1:90,2] + -34.619;
   1:L PR[91] 10mm/sec CNT100;
   1:  PR[GP1:91,1] = PR[GP1:90,1] + -37.491;
   1:  PR[GP1:91,2] = PR[GP1:90,2] + -34.696;
   1:L PR[91] 10mm/sec CNT100;
   1:  PR[GP1:91,1] = PR[GP1:90,1] + -31.930;
   1:  PR[GP1:91,2] = PR[GP1:90,2] + -33.794;
   1:L PR[91] 10mm/sec CNT100;
   1:  PR[GP1:91,1] = PR[GP1:90,1] + -26.917;
   1:  PR[GP1:91,2] = PR[GP1:90,2] + -33.059;
   1:L PR[91] 10mm/sec CNT100;
   1:  PR[GP1:91,1] = PR[GP1:90,1] + -26.057;
   1:  PR[GP1:91,2] = PR[GP1:90,2] + -32.732;
   1:L PR[91] 10mm/sec CNT100;
   1:  PR[GP1:91,1] = PR[GP1:90,1] + -17.434;
   1:  PR[GP1:91,2] = PR[GP1:90,2] + -28.526;
   1:L PR[91] 10mm/sec CNT100;
   1:  PR[GP1:91,1] = PR[GP1:90,1] + -15.094;
   1:  PR[GP1:91,2] = PR[GP1:90,2] + -26.719;
   1:L PR[91] 10mm/sec CNT100;
   1:  PR[GP1:91,1] = PR[GP1:90,1] + -9.796;
   1:  PR[GP1:91,2] = PR[GP1:90,2] + -21.603;
   1:L PR[91] 10mm/sec CNT100;
   1:  PR[GP1:91,1] = PR[GP1:90,1] + -7.037;
   1:  PR[GP1:91,2] = PR[GP1:90,2] + -17.602;
   1:L PR[91] 10mm/sec CNT100;
   1:  PR[GP1:91,1] = PR[GP1:90,1] + -4.292;
   1:  PR[GP1:91,2] = PR[GP1:90,2] + -12.348;
   1:L PR[91] 10mm/sec CNT100;
   1:  PR[GP1:91,1] = PR[GP1:90,1] + -4.162;
   1:  PR[GP1:91,2] = PR[GP1:90,2] + -12.391;
   1:L PR[91] 10mm/sec CNT100;
   1:  PR[GP1:91,1] = PR[GP1:90,1] + -3.515;
   1:  PR[GP1:91,2] = PR[GP1:90,2] + -11.683;
   1:L PR[91] 10mm/sec CNT100;
   1:  PR[GP1:91,1] = PR[GP1:90,1] + -1.653;
   1:  PR[GP1:91,2] = PR[GP1:90,2] + -9.457;
   1:L PR[91] 10mm/sec CNT100;
   1:  PR[GP1:91,1] = PR[GP1:90,1] + -0.698;
   1:  PR[GP1:91,2] = PR[GP1:90,2] + -9.531;
   1:L PR[91] 10mm/sec CNT100;
   1:  PR[GP1:91,1] = PR[GP1:90,1] + -0.692;
   1:  PR[GP1:91,2] = PR[GP1:90,2] + -9.535;
   1:L PR[91] 10mm/sec CNT100;
   1:  PR[GP1:91,1] = PR[GP1:90,1] + 2.599;
   1:  PR[GP1:91,2] = PR[GP1:90,2] + -9.501;
   1:L PR[91] 10mm/sec CNT100;
   1:  PR[GP1:91,1] = PR[GP1:90,1] + 2.957;
   1:  PR[GP1:91,2] = PR[GP1:90,2] + -10.182;
   1:L PR[91] 10mm/sec CNT100;
   1:  PR[GP1:91,1] = PR[GP1:90,1] + 3.270;
   1:  PR[GP1:91,2] = PR[GP1:90,2] + -10.543;
   1:L PR[91] 10mm/sec CNT100;
   1:  PR[GP1:91,1] = PR[GP1:90,1] + 4.310;
   1:  PR[GP1:91,2] = PR[GP1:90,2] + -11.675;
   1:L PR[91] 10mm/sec CNT100;
   1:  PR[GP1:91,1] = PR[GP1:90,1] + 5.006;
   1:  PR[GP1:91,2] = PR[GP1:90,2] + -12.508;
   1:L PR[91] 10mm/sec CNT100;
   1:  PR[GP1:91,1] = PR[GP1:90,1] + 5.270;
   1:  PR[GP1:91,2] = PR[GP1:90,2] + -12.675;
   1:L PR[91] 10mm/sec CNT100;
   1:  PR[GP1:91,1] = PR[GP1:90,1] + 7.848;
   1:  PR[GP1:91,2] = PR[GP1:90,2] + -17.580;
   1:L PR[91] 10mm/sec CNT100;
   1:  PR[GP1:91,1] = PR[GP1:90,1] + 10.611;
   1:  PR[GP1:91,2] = PR[GP1:90,2] + -21.587;
   1:L PR[91] 10mm/sec CNT100;
   1:  PR[GP1:91,1] = PR[GP1:90,1] + 15.905;
   1:  PR[GP1:91,2] = PR[GP1:90,2] + -26.713;
   1:L PR[91] 10mm/sec CNT100;
   1:  PR[GP1:91,1] = PR[GP1:90,1] + 18.245;
   1:  PR[GP1:91,2] = PR[GP1:90,2] + -28.523;
   1:L PR[91] 10mm/sec CNT100;
   1:  PR[GP1:91,1] = PR[GP1:90,1] + 26.864;
   1:  PR[GP1:91,2] = PR[GP1:90,2] + -32.726;
   1:L PR[91] 10mm/sec CNT100;
   1:  PR[GP1:91,1] = PR[GP1:90,1] + 27.725;
   1:  PR[GP1:91,2] = PR[GP1:90,2] + -33.053;
   1:L PR[91] 10mm/sec CNT100;
   1:  PR[GP1:91,1] = PR[GP1:90,1] + 32.751;
   1:  PR[GP1:91,2] = PR[GP1:90,2] + -33.793;
   1:L PR[91] 10mm/sec CNT100;
   1:  PR[GP1:91,1] = PR[GP1:90,1] + 38.301;
   1:  PR[GP1:91,2] = PR[GP1:90,2] + -34.696;
   1:L PR[91] 10mm/sec CNT100;
   1:  PR[GP1:91,1] = PR[GP1:90,1] + 39.228;
   1:  PR[GP1:91,2] = PR[GP1:90,2] + -34.620;
   1:L PR[91] 10mm/sec CNT100;
   1:  PR[GP1:91,1] = PR[GP1:90,1] + 48.952;
   1:  PR[GP1:91,2] = PR[GP1:90,2] + -33.144;
   1:L PR[91] 10mm/sec CNT100;
   1:  PR[GP1:91,1] = PR[GP1:90,1] + 51.382;
   1:  PR[GP1:91,2] = PR[GP1:90,2] + -32.088;
   1:L PR[91] 10mm/sec CNT100;
   1:  PR[GP1:91,1] = PR[GP1:90,1] + 58.784;
   1:  PR[GP1:91,2] = PR[GP1:90,2] + -28.397;
   1:L PR[91] 10mm/sec CNT100;
   1:  PR[GP1:91,1] = PR[GP1:90,1] + 61.709;
   1:  PR[GP1:91,2] = PR[GP1:90,2] + -25.728;
   1:L PR[91] 10mm/sec CNT100;
   1:  PR[GP1:91,1] = PR[GP1:90,1] + 66.748;
   1:  PR[GP1:91,2] = PR[GP1:90,2] + -20.763;
   1:L PR[91] 10mm/sec CNT100;
   1:  PR[GP1:91,1] = PR[GP1:90,1] + 69.064;
   1:  PR[GP1:91,2] = PR[GP1:90,2] + -16.524;
   1:L PR[91] 10mm/sec CNT100;
   1:  PR[GP1:91,1] = PR[GP1:90,1] + 71.936;
   1:  PR[GP1:91,2] = PR[GP1:90,2] + -10.982;
   1:L PR[91] 10mm/sec CNT100;
   1:  PR[GP1:91,1] = PR[GP1:90,1] + 72.841;
   1:  PR[GP1:91,2] = PR[GP1:90,2] + -5.632;
   1:L PR[91] 10mm/sec CNT100;
   1:  PR[GP1:91,1] = PR[GP1:90,1] + 73.742;
   1:  PR[GP1:91,2] = PR[GP1:90,2] + -0.007;
   1:L PR[91] 10mm/sec CNT100;
   1:  PR[GP1:91,1] = PR[GP1:90,1] + 72.843;
   1:  PR[GP1:91,2] = PR[GP1:90,2] + 5.297;
   1:L PR[91] 10mm/sec CNT100;
   1:  PR[GP1:91,1] = PR[GP1:90,1] + 71.935;
   1:  PR[GP1:91,2] = PR[GP1:90,2] + 10.976;
   1:L PR[91] 10mm/sec CNT100;
   1:  PR[GP1:91,1] = PR[GP1:90,1] + 69.064;
   1:  PR[GP1:91,2] = PR[GP1:90,2] + 16.515;
   1:L PR[91] 10mm/sec CNT100;
   1:  PR[GP1:91,1] = PR[GP1:90,1] + 66.748;
   1:  PR[GP1:91,2] = PR[GP1:90,2] + 20.755;
   1:L PR[91] 10mm/sec CNT100;
   1:  PR[GP1:91,1] = PR[GP1:90,1] + 61.710;
   1:  PR[GP1:91,2] = PR[GP1:90,2] + 25.719;
   1:L PR[91] 10mm/sec CNT100;
   1:  PR[GP1:91,1] = PR[GP1:90,1] + 58.784;
   1:  PR[GP1:91,2] = PR[GP1:90,2] + 28.388;
   1:L PR[91] 10mm/sec CNT100;
   1:  PR[GP1:91,1] = PR[GP1:90,1] + 51.382;
   1:  PR[GP1:91,2] = PR[GP1:90,2] + 32.079;
   1:L PR[91] 10mm/sec CNT100;
   1:  PR[GP1:91,1] = PR[GP1:90,1] + 48.952;
   1:  PR[GP1:91,2] = PR[GP1:90,2] + 33.135;
   1:L PR[91] 10mm/sec CNT100;
   1:  PR[GP1:91,1] = PR[GP1:90,1] + 39.228;
   1:  PR[GP1:91,2] = PR[GP1:90,2] + 34.611;
   1:L PR[91] 10mm/sec CNT100;
   1:  PR[GP1:91,1] = PR[GP1:90,1] + 38.301;
   1:  PR[GP1:91,2] = PR[GP1:90,2] + 34.687;
   1:L PR[91] 10mm/sec CNT100;
   1:  PR[GP1:91,1] = PR[GP1:90,1] + 32.751;
   1:  PR[GP1:91,2] = PR[GP1:90,2] + 33.784;
   1:L PR[91] 10mm/sec CNT100;
   1:  PR[GP1:91,1] = PR[GP1:90,1] + 27.725;
   1:  PR[GP1:91,2] = PR[GP1:90,2] + 33.044;
   1:L PR[91] 10mm/sec CNT100;
   1:  PR[GP1:91,1] = PR[GP1:90,1] + 26.864;
   1:  PR[GP1:91,2] = PR[GP1:90,2] + 32.717;
   1:L PR[91] 10mm/sec CNT100;
   1:  PR[GP1:91,1] = PR[GP1:90,1] + 18.245;
   1:  PR[GP1:91,2] = PR[GP1:90,2] + 28.514;
   1:L PR[91] 10mm/sec CNT100;
   1:  PR[GP1:91,1] = PR[GP1:90,1] + 15.904;
   1:  PR[GP1:91,2] = PR[GP1:90,2] + 26.704;
   1:L PR[91] 10mm/sec CNT100;
   1:  PR[GP1:91,1] = PR[GP1:90,1] + 10.611;
   1:  PR[GP1:91,2] = PR[GP1:90,2] + 21.578;
   1:L PR[91] 10mm/sec CNT100;
   1:  PR[GP1:91,1] = PR[GP1:90,1] + 7.859;
   1:  PR[GP1:91,2] = PR[GP1:90,2] + 17.592;
   1:L PR[91] 10mm/sec CNT100;
   1:  PR[GP1:91,1] = PR[GP1:90,1] + 5.308;
   1:  PR[GP1:91,2] = PR[GP1:90,2] + 12.738;
   1:L PR[91] 10mm/sec CNT100;
   1:  PR[GP1:91,1] = PR[GP1:90,1] + 4.385;
   1:  PR[GP1:91,2] = PR[GP1:90,2] + 11.747;
   1:L PR[91] 10mm/sec CNT100;
   1:  PR[GP1:91,1] = PR[GP1:90,1] + 2.846;
   1:  PR[GP1:91,2] = PR[GP1:90,2] + 9.883;
   1:L PR[91] 10mm/sec CNT100;
   1:  PR[GP1:91,1] = PR[GP1:90,1] + 2.582;
   1:  PR[GP1:91,2] = PR[GP1:90,2] + 9.595;
   1:L PR[91] 10mm/sec CNT100;
   1:  PR[GP1:91,1] = PR[GP1:90,1] + 2.293;
   1:  PR[GP1:91,2] = PR[GP1:90,2] + 9.436;
   1:L PR[91] 10mm/sec CNT100;
   1:  PR[GP1:91,1] = PR[GP1:90,1] + -1.550;
   1:  PR[GP1:91,2] = PR[GP1:90,2] + 10.608;
   1:  PR[GP1:91,3] = PR[GP1:90,3] + 27.930;
   1:L PR[91] 10mm/sec CNT100;
   1:  PR[GP1:91,1] = PR[GP1:90,1] + -1.819;
   1:  PR[GP1:91,2] = PR[GP1:90,2] + 10.765;
   1:L PR[91] 10mm/sec CNT100;
   1:  PR[GP1:91,1] = PR[GP1:90,1] + -4.498;
   1:  PR[GP1:91,2] = PR[GP1:90,2] + 13.655;
   1:L PR[91] 10mm/sec CNT100;
   1:  PR[GP1:91,1] = PR[GP1:90,1] + -4.513;
   1:  PR[GP1:91,2] = PR[GP1:90,2] + 13.790;
   1:L PR[91] 10mm/sec CNT100;
   1:  PR[GP1:91,1] = PR[GP1:90,1] + -5.933;
   1:  PR[GP1:91,2] = PR[GP1:90,2] + 16.497;
   1:L PR[91] 10mm/sec CNT100;
   1:  PR[GP1:91,1] = PR[GP1:90,1] + -9.892;
   1:  PR[GP1:91,2] = PR[GP1:90,2] + 22.231;
   1:L PR[91] 10mm/sec CNT100;
   1:  PR[GP1:91,1] = PR[GP1:90,1] + -13.671;
   1:  PR[GP1:91,2] = PR[GP1:90,2] + 25.881;
   1:L PR[91] 10mm/sec CNT100;
   1:  PR[GP1:91,1] = PR[GP1:90,1] + -17.594;
   1:  PR[GP1:91,2] = PR[GP1:90,2] + 28.910;
   1:L PR[91] 10mm/sec CNT100;
   1:  PR[GP1:91,1] = PR[GP1:90,1] + -24.399;
   1:  PR[GP1:91,2] = PR[GP1:90,2] + 32.229;
   1:L PR[91] 10mm/sec CNT100;
   1:  PR[GP1:91,1] = PR[GP1:90,1] + -27.059;
   1:  PR[GP1:91,2] = PR[GP1:90,2] + 33.240;
   1:L PR[91] 10mm/sec CNT100;
   1:  PR[GP1:91,1] = PR[GP1:90,1] + -36.940;
   1:  PR[GP1:91,2] = PR[GP1:90,2] + 34.689;
   1:L PR[91] 10mm/sec CNT100;
   1:  PR[GP1:91,1] = PR[GP1:90,1] + -37.599;
   1:  PR[GP1:91,2] = PR[GP1:90,2] + 34.736;
   1:L PR[91] 10mm/sec CNT100;
   1:  PR[GP1:91,1] = PR[GP1:90,1] + -41.544;
   1:  PR[GP1:91,2] = PR[GP1:90,2] + 34.100;
   1:L PR[91] 10mm/sec CNT100;
   1:  PR[GP1:91,1] = PR[GP1:90,1] + -48.258;
   1:  PR[GP1:91,2] = PR[GP1:90,2] + 33.081;
   1:L PR[91] 10mm/sec CNT100;
   1:  PR[GP1:91,1] = PR[GP1:90,1] + -49.210;
   1:  PR[GP1:91,2] = PR[GP1:90,2] + 32.667;
   1:L PR[91] 10mm/sec CNT100;
   1:  PR[GP1:91,1] = PR[GP1:90,1] + -57.986;
   1:  PR[GP1:91,2] = PR[GP1:90,2] + 28.284;
   1:L PR[91] 10mm/sec CNT100;
   1:  PR[GP1:91,1] = PR[GP1:90,1] + -59.805;
   1:  PR[GP1:91,2] = PR[GP1:90,2] + 26.625;
   1:L PR[91] 10mm/sec CNT100;
   1:  PR[GP1:91,1] = PR[GP1:90,1] + -65.861;
   1:  PR[GP1:91,2] = PR[GP1:90,2] + 20.664;
   1:L PR[91] 10mm/sec CNT100;
   1:  PR[GP1:91,1] = PR[GP1:90,1] + -67.504;
   1:  PR[GP1:91,2] = PR[GP1:90,2] + 17.657;
   1:L PR[91] 10mm/sec CNT100;
   1:  PR[GP1:91,1] = PR[GP1:90,1] + -70.992;
   1:  PR[GP1:91,2] = PR[GP1:90,2] + 10.906;
   1:L PR[91] 10mm/sec CNT100;
   1:  PR[GP1:91,1] = PR[GP1:90,1] + -71.668;
   1:  PR[GP1:91,2] = PR[GP1:90,2] + 6.914;
   1:L PR[91] 10mm/sec CNT100;
   1:  PR[GP1:91,1] = PR[GP1:90,1] + -72.776;
   1:  PR[GP1:91,2] = PR[GP1:90,2] + -0.002;
   1:L PR[91] 10mm/sec CNT100;
   1:  PR[GP1:91,1] = PR[GP1:90,1] + -72.094;
   1:  PR[GP1:91,2] = PR[GP1:90,2] + -4.027;
   1:L PR[91] 10mm/sec CNT100;
   1:  PR[GP1:91,1] = PR[GP1:90,1] + -70.991;
   1:  PR[GP1:91,2] = PR[GP1:90,2] + -10.918;
   1:L PR[91] 10mm/sec CNT100;
   1:  PR[GP1:91,1] = PR[GP1:90,1] + -67.504;
   1:  PR[GP1:91,2] = PR[GP1:90,2] + -17.666;
   1:L PR[91] 10mm/sec CNT100;
   1:  PR[GP1:91,1] = PR[GP1:90,1] + -65.861;
   1:  PR[GP1:91,2] = PR[GP1:90,2] + -20.673;
   1:L PR[91] 10mm/sec CNT100;
   1:  PR[GP1:91,1] = PR[GP1:90,1] + -59.805;
   1:  PR[GP1:91,2] = PR[GP1:90,2] + -26.634;
   1:L PR[91] 10mm/sec CNT100;
   1:  PR[GP1:91,1] = PR[GP1:90,1] + -57.986;
   1:  PR[GP1:91,2] = PR[GP1:90,2] + -28.293;
   1:L PR[91] 10mm/sec CNT100;
   1:  PR[GP1:91,1] = PR[GP1:90,1] + -49.210;
   1:  PR[GP1:91,2] = PR[GP1:90,2] + -32.676;
   1:L PR[91] 10mm/sec CNT100;
   1:  PR[GP1:91,1] = PR[GP1:90,1] + -48.258;
   1:  PR[GP1:91,2] = PR[GP1:90,2] + -33.089;
   1:L PR[91] 10mm/sec CNT100;
   1:  PR[GP1:91,1] = PR[GP1:90,1] + -41.544;
   1:  PR[GP1:91,2] = PR[GP1:90,2] + -34.109;
   1:L PR[91] 10mm/sec CNT100;
   1:  PR[GP1:91,1] = PR[GP1:90,1] + -37.599;
   1:  PR[GP1:91,2] = PR[GP1:90,2] + -34.745;
   1:L PR[91] 10mm/sec CNT100;
   1:  PR[GP1:91,1] = PR[GP1:90,1] + -36.940;
   1:  PR[GP1:91,2] = PR[GP1:90,2] + -34.698;
   1:L PR[91] 10mm/sec CNT100;
   1:  PR[GP1:91,1] = PR[GP1:90,1] + -27.059;
   1:  PR[GP1:91,2] = PR[GP1:90,2] + -33.249;
   1:L PR[91] 10mm/sec CNT100;
   1:  PR[GP1:91,1] = PR[GP1:90,1] + -24.399;
   1:  PR[GP1:91,2] = PR[GP1:90,2] + -32.238;
   1:L PR[91] 10mm/sec CNT100;
   1:  PR[GP1:91,1] = PR[GP1:90,1] + -17.594;
   1:  PR[GP1:91,2] = PR[GP1:90,2] + -28.918;
   1:L PR[91] 10mm/sec CNT100;
   1:  PR[GP1:91,1] = PR[GP1:90,1] + -13.671;
   1:  PR[GP1:91,2] = PR[GP1:90,2] + -25.889;
   1:L PR[91] 10mm/sec CNT100;
   1:  PR[GP1:91,1] = PR[GP1:90,1] + -9.892;
   1:  PR[GP1:91,2] = PR[GP1:90,2] + -22.240;
   1:L PR[91] 10mm/sec CNT100;
   1:  PR[GP1:91,1] = PR[GP1:90,1] + -5.918;
   1:  PR[GP1:91,2] = PR[GP1:90,2] + -16.477;
   1:L PR[91] 10mm/sec CNT100;
   1:  PR[GP1:91,1] = PR[GP1:90,1] + -4.222;
   1:  PR[GP1:91,2] = PR[GP1:90,2] + -13.232;
   1:L PR[91] 10mm/sec CNT100;
   1:  PR[GP1:91,1] = PR[GP1:90,1] + -4.099;
   1:  PR[GP1:91,2] = PR[GP1:90,2] + -13.273;
   1:L PR[91] 10mm/sec CNT100;
   1:  PR[GP1:91,1] = PR[GP1:90,1] + -1.821;
   1:  PR[GP1:91,2] = PR[GP1:90,2] + -10.775;
   1:L PR[91] 10mm/sec CNT100;
   1:  PR[GP1:91,1] = PR[GP1:90,1] + -1.551;
   1:  PR[GP1:91,2] = PR[GP1:90,2] + -10.617;
   1:L PR[91] 10mm/sec CNT100;
   1:  PR[GP1:91,1] = PR[GP1:90,1] + 2.408;
   1:  PR[GP1:91,2] = PR[GP1:90,2] + -10.578;
   1:L PR[91] 10mm/sec CNT100;
   1:  PR[GP1:91,1] = PR[GP1:90,1] + 4.539;
   1:  PR[GP1:91,2] = PR[GP1:90,2] + -13.130;
   1:L PR[91] 10mm/sec CNT100;
   1:  PR[GP1:91,1] = PR[GP1:90,1] + 5.200;
   1:  PR[GP1:91,2] = PR[GP1:90,2] + -13.547;
   1:L PR[91] 10mm/sec CNT100;
   1:  PR[GP1:91,1] = PR[GP1:90,1] + 6.729;
   1:  PR[GP1:91,2] = PR[GP1:90,2] + -16.458;
   1:L PR[91] 10mm/sec CNT100;
   1:  PR[GP1:91,1] = PR[GP1:90,1] + 10.709;
   1:  PR[GP1:91,2] = PR[GP1:90,2] + -22.228;
   1:L PR[91] 10mm/sec CNT100;
   1:  PR[GP1:91,1] = PR[GP1:90,1] + 14.485;
   1:  PR[GP1:91,2] = PR[GP1:90,2] + -25.884;
   1:L PR[91] 10mm/sec CNT100;
   1:  PR[GP1:91,1] = PR[GP1:90,1] + 18.407;
   1:  PR[GP1:91,2] = PR[GP1:90,2] + -28.917;
   1:L PR[91] 10mm/sec CNT100;
   1:  PR[GP1:91,1] = PR[GP1:90,1] + 25.209;
   1:  PR[GP1:91,2] = PR[GP1:90,2] + -32.234;
   1:L PR[91] 10mm/sec CNT100;
   1:  PR[GP1:91,1] = PR[GP1:90,1] + 27.870;
   1:  PR[GP1:91,2] = PR[GP1:90,2] + -33.244;
   1:L PR[91] 10mm/sec CNT100;
   1:  PR[GP1:91,1] = PR[GP1:90,1] + 37.749;
   1:  PR[GP1:91,2] = PR[GP1:90,2] + -34.698;
   1:L PR[91] 10mm/sec CNT100;
   1:  PR[GP1:91,1] = PR[GP1:90,1] + 38.409;
   1:  PR[GP1:91,2] = PR[GP1:90,2] + -34.745;
   1:L PR[91] 10mm/sec CNT100;
   1:  PR[GP1:91,1] = PR[GP1:90,1] + 42.365;
   1:  PR[GP1:91,2] = PR[GP1:90,2] + -34.108;
   1:L PR[91] 10mm/sec CNT100;
   1:  PR[GP1:91,1] = PR[GP1:90,1] + 49.071;
   1:  PR[GP1:91,2] = PR[GP1:90,2] + -33.090;
   1:L PR[91] 10mm/sec CNT100;
   1:  PR[GP1:91,1] = PR[GP1:90,1] + 50.021;
   1:  PR[GP1:91,2] = PR[GP1:90,2] + -32.677;
   1:L PR[91] 10mm/sec CNT100;
   1:  PR[GP1:91,1] = PR[GP1:90,1] + 58.802;
   1:  PR[GP1:91,2] = PR[GP1:90,2] + -28.299;
   1:L PR[91] 10mm/sec CNT100;
   1:  PR[GP1:91,1] = PR[GP1:90,1] + 60.620;
   1:  PR[GP1:91,2] = PR[GP1:90,2] + -26.640;
   1:L PR[91] 10mm/sec CNT100;
   1:  PR[GP1:91,1] = PR[GP1:90,1] + 66.680;
   1:  PR[GP1:91,2] = PR[GP1:90,2] + -20.669;
   1:L PR[91] 10mm/sec CNT100;
   1:  PR[GP1:91,1] = PR[GP1:90,1] + 68.322;
   1:  PR[GP1:91,2] = PR[GP1:90,2] + -17.663;
   1:L PR[91] 10mm/sec CNT100;
   1:  PR[GP1:91,1] = PR[GP1:90,1] + 71.812;
   1:  PR[GP1:91,2] = PR[GP1:90,2] + -10.928;
   1:L PR[91] 10mm/sec CNT100;
   1:  PR[GP1:91,1] = PR[GP1:90,1] + 72.488;
   1:  PR[GP1:91,2] = PR[GP1:90,2] + -6.935;
   1:L PR[91] 10mm/sec CNT100;
   1:  PR[GP1:91,1] = PR[GP1:90,1] + 73.597;
   1:  PR[GP1:91,2] = PR[GP1:90,2] + -0.007;
   1:L PR[91] 10mm/sec CNT100;
   1:  PR[GP1:91,1] = PR[GP1:90,1] + 72.914;
   1:  PR[GP1:91,2] = PR[GP1:90,2] + 4.020;
   1:L PR[91] 10mm/sec CNT100;
   1:  PR[GP1:91,1] = PR[GP1:90,1] + 71.811;
   1:  PR[GP1:91,2] = PR[GP1:90,2] + 10.922;
   1:L PR[91] 10mm/sec CNT100;
   1:  PR[GP1:91,1] = PR[GP1:90,1] + 68.322;
   1:  PR[GP1:91,2] = PR[GP1:90,2] + 17.654;
   1:L PR[91] 10mm/sec CNT100;
   1:  PR[GP1:91,1] = PR[GP1:90,1] + 66.680;
   1:  PR[GP1:91,2] = PR[GP1:90,2] + 20.660;
   1:L PR[91] 10mm/sec CNT100;
   1:  PR[GP1:91,1] = PR[GP1:90,1] + 60.620;
   1:  PR[GP1:91,2] = PR[GP1:90,2] + 26.631;
   1:L PR[91] 10mm/sec CNT100;
   1:  PR[GP1:91,1] = PR[GP1:90,1] + 58.802;
   1:  PR[GP1:91,2] = PR[GP1:90,2] + 28.290;
   1:L PR[91] 10mm/sec CNT100;
   1:  PR[GP1:91,1] = PR[GP1:90,1] + 50.021;
   1:  PR[GP1:91,2] = PR[GP1:90,2] + 32.668;
   1:L PR[91] 10mm/sec CNT100;
   1:  PR[GP1:91,1] = PR[GP1:90,1] + 49.071;
   1:  PR[GP1:91,2] = PR[GP1:90,2] + 33.081;
   1:L PR[91] 10mm/sec CNT100;
   1:  PR[GP1:91,1] = PR[GP1:90,1] + 42.365;
   1:  PR[GP1:91,2] = PR[GP1:90,2] + 34.099;
   1:L PR[91] 10mm/sec CNT100;
   1:  PR[GP1:91,1] = PR[GP1:90,1] + 38.409;
   1:  PR[GP1:91,2] = PR[GP1:90,2] + 34.736;
   1:L PR[91] 10mm/sec CNT100;
   1:  PR[GP1:91,1] = PR[GP1:90,1] + 37.748;
   1:  PR[GP1:91,2] = PR[GP1:90,2] + 34.689;
   1:L PR[91] 10mm/sec CNT100;
   1:  PR[GP1:91,1] = PR[GP1:90,1] + 27.870;
   1:  PR[GP1:91,2] = PR[GP1:90,2] + 33.235;
   1:L PR[91] 10mm/sec CNT100;
   1:  PR[GP1:91,1] = PR[GP1:90,1] + 25.209;
   1:  PR[GP1:91,2] = PR[GP1:90,2] + 32.225;
   1:L PR[91] 10mm/sec CNT100;
   1:  PR[GP1:91,1] = PR[GP1:90,1] + 18.407;
   1:  PR[GP1:91,2] = PR[GP1:90,2] + 28.908;
   1:L PR[91] 10mm/sec CNT100;
   1:  PR[GP1:91,1] = PR[GP1:90,1] + 14.485;
   1:  PR[GP1:91,2] = PR[GP1:90,2] + 25.876;
   1:L PR[91] 10mm/sec CNT100;
   1:  PR[GP1:91,1] = PR[GP1:90,1] + 10.709;
   1:  PR[GP1:91,2] = PR[GP1:90,2] + 22.219;
   1:L PR[91] 10mm/sec CNT100;
   1:  PR[GP1:91,1] = PR[GP1:90,1] + 6.745;
   1:  PR[GP1:91,2] = PR[GP1:90,2] + 16.478;
   1:L PR[91] 10mm/sec CNT100;
   1:  PR[GP1:91,1] = PR[GP1:90,1] + 5.238;
   1:  PR[GP1:91,2] = PR[GP1:90,2] + 13.610;
   1:L PR[91] 10mm/sec CNT100;
   1:  PR[GP1:91,1] = PR[GP1:90,1] + 2.557;
   1:  PR[GP1:91,2] = PR[GP1:90,2] + 10.726;
   1:L PR[91] 10mm/sec CNT100;
   1:  PR[GP1:91,1] = PR[GP1:90,1] + 2.290;
   1:  PR[GP1:91,2] = PR[GP1:90,2] + 10.570;
   1:L PR[91] 10mm/sec CNT100;
   1:  PR[GP1:91,1] = PR[GP1:90,1] + -1.325;
   1:  PR[GP1:91,2] = PR[GP1:90,2] + 11.527;
   1:  PR[GP1:91,3] = PR[GP1:90,3] + 29.260;
   1:L PR[91] 10mm/sec CNT100;
   1:  PR[GP1:91,1] = PR[GP1:90,1] + -2.087;
   1:  PR[GP1:91,2] = PR[GP1:90,2] + 11.973;
   1:L PR[91] 10mm/sec CNT100;
   1:  PR[GP1:91,1] = PR[GP1:90,1] + -4.423;
   1:  PR[GP1:91,2] = PR[GP1:90,2] + 14.493;
   1:L PR[91] 10mm/sec CNT100;
   1:  PR[GP1:91,1] = PR[GP1:90,1] + -4.442;
   1:  PR[GP1:91,2] = PR[GP1:90,2] + 14.662;
   1:L PR[91] 10mm/sec CNT100;
   1:  PR[GP1:91,1] = PR[GP1:90,1] + -4.819;
   1:  PR[GP1:91,2] = PR[GP1:90,2] + 15.381;
   1:L PR[91] 10mm/sec CNT100;
   1:  PR[GP1:91,1] = PR[GP1:90,1] + -9.988;
   1:  PR[GP1:91,2] = PR[GP1:90,2] + 22.869;
   1:L PR[91] 10mm/sec CNT100;
   1:  PR[GP1:91,1] = PR[GP1:90,1] + -12.248;
   1:  PR[GP1:91,2] = PR[GP1:90,2] + 25.051;
   1:L PR[91] 10mm/sec CNT100;
   1:  PR[GP1:91,1] = PR[GP1:90,1] + -17.754;
   1:  PR[GP1:91,2] = PR[GP1:90,2] + 29.302;
   1:L PR[91] 10mm/sec CNT100;
   1:  PR[GP1:91,1] = PR[GP1:90,1] + -22.741;
   1:  PR[GP1:91,2] = PR[GP1:90,2] + 31.734;
   1:L PR[91] 10mm/sec CNT100;
   1:  PR[GP1:91,1] = PR[GP1:90,1] + -27.202;
   1:  PR[GP1:91,2] = PR[GP1:90,2] + 33.430;
   1:L PR[91] 10mm/sec CNT100;
   1:  PR[GP1:91,1] = PR[GP1:90,1] + -35.197;
   1:  PR[GP1:91,2] = PR[GP1:90,2] + 34.603;
   1:L PR[91] 10mm/sec CNT100;
   1:  PR[GP1:91,1] = PR[GP1:90,1] + -37.673;
   1:  PR[GP1:91,2] = PR[GP1:90,2] + 34.779;
   1:L PR[91] 10mm/sec CNT100;
   1:  PR[GP1:91,1] = PR[GP1:90,1] + -47.896;
   1:  PR[GP1:91,2] = PR[GP1:90,2] + 33.132;
   1:L PR[91] 10mm/sec CNT100;
   1:  PR[GP1:91,1] = PR[GP1:90,1] + -48.302;
   1:  PR[GP1:91,2] = PR[GP1:90,2] + 33.041;
   1:L PR[91] 10mm/sec CNT100;
   1:  PR[GP1:91,1] = PR[GP1:90,1] + -58.004;
   1:  PR[GP1:91,2] = PR[GP1:90,2] + 28.186;
   1:L PR[91] 10mm/sec CNT100;
   1:  PR[GP1:91,1] = PR[GP1:90,1] + -58.716;
   1:  PR[GP1:91,2] = PR[GP1:90,2] + 27.536;
   1:L PR[91] 10mm/sec CNT100;
   1:  PR[GP1:91,1] = PR[GP1:90,1] + -65.794;
   1:  PR[GP1:91,2] = PR[GP1:90,2] + 20.570;
   1:L PR[91] 10mm/sec CNT100;
   1:  PR[GP1:91,1] = PR[GP1:90,1] + -66.762;
   1:  PR[GP1:91,2] = PR[GP1:90,2] + 18.797;
   1:L PR[91] 10mm/sec CNT100;
   1:  PR[GP1:91,1] = PR[GP1:90,1] + -70.868;
   1:  PR[GP1:91,2] = PR[GP1:90,2] + 10.851;
   1:L PR[91] 10mm/sec CNT100;
   1:  PR[GP1:91,1] = PR[GP1:90,1] + -71.315;
   1:  PR[GP1:91,2] = PR[GP1:90,2] + 8.215;
   1:L PR[91] 10mm/sec CNT100;
   1:  PR[GP1:91,1] = PR[GP1:90,1] + -72.631;
   1:  PR[GP1:91,2] = PR[GP1:90,2] + -0.002;
   1:L PR[91] 10mm/sec CNT100;
   1:  PR[GP1:91,1] = PR[GP1:90,1] + -72.165;
   1:  PR[GP1:91,2] = PR[GP1:90,2] + -2.752;
   1:L PR[91] 10mm/sec CNT100;
   1:  PR[GP1:91,1] = PR[GP1:90,1] + -70.867;
   1:  PR[GP1:91,2] = PR[GP1:90,2] + -10.862;
   1:L PR[91] 10mm/sec CNT100;
   1:  PR[GP1:91,1] = PR[GP1:90,1] + -66.762;
   1:  PR[GP1:91,2] = PR[GP1:90,2] + -18.806;
   1:L PR[91] 10mm/sec CNT100;
   1:  PR[GP1:91,1] = PR[GP1:90,1] + -65.794;
   1:  PR[GP1:91,2] = PR[GP1:90,2] + -20.579;
   1:L PR[91] 10mm/sec CNT100;
   1:  PR[GP1:91,1] = PR[GP1:90,1] + -58.716;
   1:  PR[GP1:91,2] = PR[GP1:90,2] + -27.545;
   1:L PR[91] 10mm/sec CNT100;
   1:  PR[GP1:91,1] = PR[GP1:90,1] + -58.004;
   1:  PR[GP1:91,2] = PR[GP1:90,2] + -28.194;
   1:L PR[91] 10mm/sec CNT100;
   1:  PR[GP1:91,1] = PR[GP1:90,1] + -48.302;
   1:  PR[GP1:91,2] = PR[GP1:90,2] + -33.050;
   1:L PR[91] 10mm/sec CNT100;
   1:  PR[GP1:91,1] = PR[GP1:90,1] + -47.896;
   1:  PR[GP1:91,2] = PR[GP1:90,2] + -33.141;
   1:L PR[91] 10mm/sec CNT100;
   1:  PR[GP1:91,1] = PR[GP1:90,1] + -37.673;
   1:  PR[GP1:91,2] = PR[GP1:90,2] + -34.788;
   1:L PR[91] 10mm/sec CNT100;
   1:  PR[GP1:91,1] = PR[GP1:90,1] + -35.197;
   1:  PR[GP1:91,2] = PR[GP1:90,2] + -34.612;
   1:L PR[91] 10mm/sec CNT100;
   1:  PR[GP1:91,1] = PR[GP1:90,1] + -27.202;
   1:  PR[GP1:91,2] = PR[GP1:90,2] + -33.439;
   1:L PR[91] 10mm/sec CNT100;
   1:  PR[GP1:91,1] = PR[GP1:90,1] + -22.741;
   1:  PR[GP1:91,2] = PR[GP1:90,2] + -31.743;
   1:L PR[91] 10mm/sec CNT100;
   1:  PR[GP1:91,1] = PR[GP1:90,1] + -17.754;
   1:  PR[GP1:91,2] = PR[GP1:90,2] + -29.311;
   1:L PR[91] 10mm/sec CNT100;
   1:  PR[GP1:91,1] = PR[GP1:90,1] + -12.248;
   1:  PR[GP1:91,2] = PR[GP1:90,2] + -25.060;
   1:L PR[91] 10mm/sec CNT100;
   1:  PR[GP1:91,1] = PR[GP1:90,1] + -9.989;
   1:  PR[GP1:91,2] = PR[GP1:90,2] + -22.877;
   1:L PR[91] 10mm/sec CNT100;
   1:  PR[GP1:91,1] = PR[GP1:90,1] + -4.799;
   1:  PR[GP1:91,2] = PR[GP1:90,2] + -15.352;
   1:L PR[91] 10mm/sec CNT100;
   1:  PR[GP1:91,1] = PR[GP1:90,1] + -4.352;
   1:  PR[GP1:91,2] = PR[GP1:90,2] + -14.498;
   1:L PR[91] 10mm/sec CNT100;
   1:  PR[GP1:91,1] = PR[GP1:90,1] + -3.625;
   1:  PR[GP1:91,2] = PR[GP1:90,2] + -13.705;
   1:L PR[91] 10mm/sec CNT100;
   1:  PR[GP1:91,1] = PR[GP1:90,1] + -2.092;
   1:  PR[GP1:91,2] = PR[GP1:90,2] + -11.985;
   1:L PR[91] 10mm/sec CNT100;
   1:  PR[GP1:91,1] = PR[GP1:90,1] + -1.325;
   1:  PR[GP1:91,2] = PR[GP1:90,2] + -11.536;
   1:L PR[91] 10mm/sec CNT100;
   1:  PR[GP1:91,1] = PR[GP1:90,1] + 2.194;
   1:  PR[GP1:91,2] = PR[GP1:90,2] + -11.502;
   1:L PR[91] 10mm/sec CNT100;
   1:  PR[GP1:91,1] = PR[GP1:90,1] + 4.072;
   1:  PR[GP1:91,2] = PR[GP1:90,2] + -13.753;
   1:L PR[91] 10mm/sec CNT100;
   1:  PR[GP1:91,1] = PR[GP1:90,1] + 5.130;
   1:  PR[GP1:91,2] = PR[GP1:90,2] + -14.419;
   1:L PR[91] 10mm/sec CNT100;
   1:  PR[GP1:91,1] = PR[GP1:90,1] + 5.611;
   1:  PR[GP1:91,2] = PR[GP1:90,2] + -15.335;
   1:L PR[91] 10mm/sec CNT100;
   1:  PR[GP1:91,1] = PR[GP1:90,1] + 10.807;
   1:  PR[GP1:91,2] = PR[GP1:90,2] + -22.869;
   1:L PR[91] 10mm/sec CNT100;
   1:  PR[GP1:91,1] = PR[GP1:90,1] + 13.065;
   1:  PR[GP1:91,2] = PR[GP1:90,2] + -25.056;
   1:L PR[91] 10mm/sec CNT100;
   1:  PR[GP1:91,1] = PR[GP1:90,1] + 18.569;
   1:  PR[GP1:91,2] = PR[GP1:90,2] + -29.310;
   1:L PR[91] 10mm/sec CNT100;
   1:  PR[GP1:91,1] = PR[GP1:90,1] + 23.554;
   1:  PR[GP1:91,2] = PR[GP1:90,2] + -31.741;
   1:L PR[91] 10mm/sec CNT100;
   1:  PR[GP1:91,1] = PR[GP1:90,1] + 28.015;
   1:  PR[GP1:91,2] = PR[GP1:90,2] + -33.435;
   1:L PR[91] 10mm/sec CNT100;
   1:  PR[GP1:91,1] = PR[GP1:90,1] + 36.007;
   1:  PR[GP1:91,2] = PR[GP1:90,2] + -34.611;
   1:L PR[91] 10mm/sec CNT100;
   1:  PR[GP1:91,1] = PR[GP1:90,1] + 38.485;
   1:  PR[GP1:91,2] = PR[GP1:90,2] + -34.788;
   1:L PR[91] 10mm/sec CNT100;
   1:  PR[GP1:91,1] = PR[GP1:90,1] + 48.707;
   1:  PR[GP1:91,2] = PR[GP1:90,2] + -33.142;
   1:L PR[91] 10mm/sec CNT100;
   1:  PR[GP1:91,1] = PR[GP1:90,1] + 49.114;
   1:  PR[GP1:91,2] = PR[GP1:90,2] + -33.050;
   1:L PR[91] 10mm/sec CNT100;
   1:  PR[GP1:91,1] = PR[GP1:90,1] + 58.819;
   1:  PR[GP1:91,2] = PR[GP1:90,2] + -28.201;
   1:L PR[91] 10mm/sec CNT100;
   1:  PR[GP1:91,1] = PR[GP1:90,1] + 59.531;
   1:  PR[GP1:91,2] = PR[GP1:90,2] + -27.552;
   1:L PR[91] 10mm/sec CNT100;
   1:  PR[GP1:91,1] = PR[GP1:90,1] + 66.612;
   1:  PR[GP1:91,2] = PR[GP1:90,2] + -20.574;
   1:L PR[91] 10mm/sec CNT100;
   1:  PR[GP1:91,1] = PR[GP1:90,1] + 67.580;
   1:  PR[GP1:91,2] = PR[GP1:90,2] + -18.802;
   1:L PR[91] 10mm/sec CNT100;
   1:  PR[GP1:91,1] = PR[GP1:90,1] + 71.688;
   1:  PR[GP1:91,2] = PR[GP1:90,2] + -10.875;
   1:L PR[91] 10mm/sec CNT100;
   1:  PR[GP1:91,1] = PR[GP1:90,1] + 72.135;
   1:  PR[GP1:91,2] = PR[GP1:90,2] + -8.237;
   1:L PR[91] 10mm/sec CNT100;
   1:  PR[GP1:91,1] = PR[GP1:90,1] + 73.452;
   1:  PR[GP1:91,2] = PR[GP1:90,2] + -0.007;
   1:L PR[91] 10mm/sec CNT100;
   1:  PR[GP1:91,1] = PR[GP1:90,1] + 72.986;
   1:  PR[GP1:91,2] = PR[GP1:90,2] + 2.744;
   1:L PR[91] 10mm/sec CNT100;
   1:  PR[GP1:91,1] = PR[GP1:90,1] + 71.687;
   1:  PR[GP1:91,2] = PR[GP1:90,2] + 10.868;
   1:L PR[91] 10mm/sec CNT100;
   1:  PR[GP1:91,1] = PR[GP1:90,1] + 67.580;
   1:  PR[GP1:91,2] = PR[GP1:90,2] + 18.793;
   1:L PR[91] 10mm/sec CNT100;
   1:  PR[GP1:91,1] = PR[GP1:90,1] + 66.612;
   1:  PR[GP1:91,2] = PR[GP1:90,2] + 20.565;
   1:L PR[91] 10mm/sec CNT100;
   1:  PR[GP1:91,1] = PR[GP1:90,1] + 59.531;
   1:  PR[GP1:91,2] = PR[GP1:90,2] + 27.543;
   1:L PR[91] 10mm/sec CNT100;
   1:  PR[GP1:91,1] = PR[GP1:90,1] + 58.819;
   1:  PR[GP1:91,2] = PR[GP1:90,2] + 28.193;
   1:L PR[91] 10mm/sec CNT100;
   1:  PR[GP1:91,1] = PR[GP1:90,1] + 49.114;
   1:  PR[GP1:91,2] = PR[GP1:90,2] + 33.041;
   1:L PR[91] 10mm/sec CNT100;
   1:  PR[GP1:91,1] = PR[GP1:90,1] + 48.707;
   1:  PR[GP1:91,2] = PR[GP1:90,2] + 33.133;
   1:L PR[91] 10mm/sec CNT100;
   1:  PR[GP1:91,1] = PR[GP1:90,1] + 38.485;
   1:  PR[GP1:91,2] = PR[GP1:90,2] + 34.779;
   1:L PR[91] 10mm/sec CNT100;
   1:  PR[GP1:91,1] = PR[GP1:90,1] + 36.007;
   1:  PR[GP1:91,2] = PR[GP1:90,2] + 34.602;
   1:L PR[91] 10mm/sec CNT100;
   1:  PR[GP1:91,1] = PR[GP1:90,1] + 28.015;
   1:  PR[GP1:91,2] = PR[GP1:90,2] + 33.426;
   1:L PR[91] 10mm/sec CNT100;
   1:  PR[GP1:91,1] = PR[GP1:90,1] + 23.554;
   1:  PR[GP1:91,2] = PR[GP1:90,2] + 31.732;
   1:L PR[91] 10mm/sec CNT100;
   1:  PR[GP1:91,1] = PR[GP1:90,1] + 18.569;
   1:  PR[GP1:91,2] = PR[GP1:90,2] + 29.302;
   1:L PR[91] 10mm/sec CNT100;
   1:  PR[GP1:91,1] = PR[GP1:90,1] + 13.065;
   1:  PR[GP1:91,2] = PR[GP1:90,2] + 25.047;
   1:L PR[91] 10mm/sec CNT100;
   1:  PR[GP1:91,1] = PR[GP1:90,1] + 10.807;
   1:  PR[GP1:91,2] = PR[GP1:90,2] + 22.860;
   1:L PR[91] 10mm/sec CNT100;
   1:  PR[GP1:91,1] = PR[GP1:90,1] + 5.631;
   1:  PR[GP1:91,2] = PR[GP1:90,2] + 15.365;
   1:L PR[91] 10mm/sec CNT100;
   1:  PR[GP1:91,1] = PR[GP1:90,1] + 5.168;
   1:  PR[GP1:91,2] = PR[GP1:90,2] + 14.484;
   1:L PR[91] 10mm/sec CNT100;
   1:  PR[GP1:91,1] = PR[GP1:90,1] + 2.840;
   1:  PR[GP1:91,2] = PR[GP1:90,2] + 11.941;
   1:L PR[91] 10mm/sec CNT100;
   1:  PR[GP1:91,1] = PR[GP1:90,1] + 2.075;
   1:  PR[GP1:91,2] = PR[GP1:90,2] + 11.494;
   1:L PR[91] 10mm/sec CNT100;
   1:  PR[GP1:91,1] = PR[GP1:90,1] + -1.099;
   1:  PR[GP1:91,2] = PR[GP1:90,2] + 12.447;
   1:  PR[GP1:91,3] = PR[GP1:90,3] + 30.590;
   1:L PR[91] 10mm/sec CNT100;
   1:  PR[GP1:91,1] = PR[GP1:90,1] + -2.354;
   1:  PR[GP1:91,2] = PR[GP1:90,2] + 13.181;
   1:L PR[91] 10mm/sec CNT100;
   1:  PR[GP1:91,1] = PR[GP1:90,1] + -4.347;
   1:  PR[GP1:91,2] = PR[GP1:90,2] + 15.331;
   1:L PR[91] 10mm/sec CNT100;
   1:  PR[GP1:91,1] = PR[GP1:90,1] + -4.362;
   1:  PR[GP1:91,2] = PR[GP1:90,2] + 15.459;
   1:L PR[91] 10mm/sec CNT100;
   1:  PR[GP1:91,1] = PR[GP1:90,1] + -7.347;
   1:  PR[GP1:91,2] = PR[GP1:90,2] + 19.541;
   1:L PR[91] 10mm/sec CNT100;
   1:  PR[GP1:91,1] = PR[GP1:90,1] + -10.085;
   1:  PR[GP1:91,2] = PR[GP1:90,2] + 23.506;
   1:L PR[91] 10mm/sec CNT100;
   1:  PR[GP1:91,1] = PR[GP1:90,1] + -10.826;
   1:  PR[GP1:91,2] = PR[GP1:90,2] + 24.221;
   1:L PR[91] 10mm/sec CNT100;
   1:  PR[GP1:91,1] = PR[GP1:90,1] + -17.914;
   1:  PR[GP1:91,2] = PR[GP1:90,2] + 29.694;
   1:L PR[91] 10mm/sec CNT100;
   1:  PR[GP1:91,1] = PR[GP1:90,1] + -21.083;
   1:  PR[GP1:91,2] = PR[GP1:90,2] + 31.240;
   1:L PR[91] 10mm/sec CNT100;
   1:  PR[GP1:91,1] = PR[GP1:90,1] + -27.345;
   1:  PR[GP1:91,2] = PR[GP1:90,2] + 33.620;
   1:L PR[91] 10mm/sec CNT100;
   1:  PR[GP1:91,1] = PR[GP1:90,1] + -33.453;
   1:  PR[GP1:91,2] = PR[GP1:90,2] + 34.516;
   1:L PR[91] 10mm/sec CNT100;
   1:  PR[GP1:91,1] = PR[GP1:90,1] + -37.748;
   1:  PR[GP1:91,2] = PR[GP1:90,2] + 34.822;
   1:L PR[91] 10mm/sec CNT100;
   1:  PR[GP1:91,1] = PR[GP1:90,1] + -46.220;
   1:  PR[GP1:91,2] = PR[GP1:90,2] + 33.456;
   1:L PR[91] 10mm/sec CNT100;
   1:  PR[GP1:91,1] = PR[GP1:90,1] + -48.284;
   1:  PR[GP1:91,2] = PR[GP1:90,2] + 32.994;
   1:L PR[91] 10mm/sec CNT100;
   1:  PR[GP1:91,1] = PR[GP1:90,1] + -57.644;
   1:  PR[GP1:91,2] = PR[GP1:90,2] + 28.287;
   1:L PR[91] 10mm/sec CNT100;
   1:  PR[GP1:91,1] = PR[GP1:90,1] + -57.963;
   1:  PR[GP1:91,2] = PR[GP1:90,2] + 28.107;
   1:L PR[91] 10mm/sec CNT100;
   1:  PR[GP1:91,1] = PR[GP1:90,1] + -65.726;
   1:  PR[GP1:91,2] = PR[GP1:90,2] + 20.476;
   1:L PR[91] 10mm/sec CNT100;
   1:  PR[GP1:91,1] = PR[GP1:90,1] + -66.020;
   1:  PR[GP1:91,2] = PR[GP1:90,2] + 19.937;
   1:L PR[91] 10mm/sec CNT100;
   1:  PR[GP1:91,1] = PR[GP1:90,1] + -70.745;
   1:  PR[GP1:91,2] = PR[GP1:90,2] + 10.796;
   1:L PR[91] 10mm/sec CNT100;
   1:  PR[GP1:91,1] = PR[GP1:90,1] + -70.961;
   1:  PR[GP1:91,2] = PR[GP1:90,2] + 9.515;
   1:L PR[91] 10mm/sec CNT100;
   1:  PR[GP1:91,1] = PR[GP1:90,1] + -72.487;
   1:  PR[GP1:91,2] = PR[GP1:90,2] + -0.002;
   1:L PR[91] 10mm/sec CNT100;
   1:  PR[GP1:91,1] = PR[GP1:90,1] + -72.237;
   1:  PR[GP1:91,2] = PR[GP1:90,2] + -1.476;
   1:L PR[91] 10mm/sec CNT100;
   1:  PR[GP1:91,1] = PR[GP1:90,1] + -70.743;
   1:  PR[GP1:91,2] = PR[GP1:90,2] + -10.807;
   1:L PR[91] 10mm/sec CNT100;
   1:  PR[GP1:91,1] = PR[GP1:90,1] + -66.020;
   1:  PR[GP1:91,2] = PR[GP1:90,2] + -19.946;
   1:L PR[91] 10mm/sec CNT100;
   1:  PR[GP1:91,1] = PR[GP1:90,1] + -65.726;
   1:  PR[GP1:91,2] = PR[GP1:90,2] + -20.485;
   1:L PR[91] 10mm/sec CNT100;
   1:  PR[GP1:91,1] = PR[GP1:90,1] + -57.963;
   1:  PR[GP1:91,2] = PR[GP1:90,2] + -28.116;
   1:L PR[91] 10mm/sec CNT100;
   1:  PR[GP1:91,1] = PR[GP1:90,1] + -57.644;
   1:  PR[GP1:91,2] = PR[GP1:90,2] + -28.296;
   1:L PR[91] 10mm/sec CNT100;
   1:  PR[GP1:91,1] = PR[GP1:90,1] + -48.284;
   1:  PR[GP1:91,2] = PR[GP1:90,2] + -33.003;
   1:L PR[91] 10mm/sec CNT100;
   1:  PR[GP1:91,1] = PR[GP1:90,1] + -46.220;
   1:  PR[GP1:91,2] = PR[GP1:90,2] + -33.465;
   1:L PR[91] 10mm/sec CNT100;
   1:  PR[GP1:91,1] = PR[GP1:90,1] + -37.748;
   1:  PR[GP1:91,2] = PR[GP1:90,2] + -34.830;
   1:L PR[91] 10mm/sec CNT100;
   1:  PR[GP1:91,1] = PR[GP1:90,1] + -33.453;
   1:  PR[GP1:91,2] = PR[GP1:90,2] + -34.525;
   1:L PR[91] 10mm/sec CNT100;
   1:  PR[GP1:91,1] = PR[GP1:90,1] + -27.345;
   1:  PR[GP1:91,2] = PR[GP1:90,2] + -33.629;
   1:L PR[91] 10mm/sec CNT100;
   1:  PR[GP1:91,1] = PR[GP1:90,1] + -21.083;
   1:  PR[GP1:91,2] = PR[GP1:90,2] + -31.249;
   1:L PR[91] 10mm/sec CNT100;
   1:  PR[GP1:91,1] = PR[GP1:90,1] + -17.914;
   1:  PR[GP1:91,2] = PR[GP1:90,2] + -29.703;
   1:L PR[91] 10mm/sec CNT100;
   1:  PR[GP1:91,1] = PR[GP1:90,1] + -10.825;
   1:  PR[GP1:91,2] = PR[GP1:90,2] + -24.230;
   1:L PR[91] 10mm/sec CNT100;
   1:  PR[GP1:91,1] = PR[GP1:90,1] + -10.085;
   1:  PR[GP1:91,2] = PR[GP1:90,2] + -23.515;
   1:L PR[91] 10mm/sec CNT100;
   1:  PR[GP1:91,1] = PR[GP1:90,1] + -7.402;
   1:  PR[GP1:91,2] = PR[GP1:90,2] + -19.624;
   1:L PR[91] 10mm/sec CNT100;
   1:  PR[GP1:91,1] = PR[GP1:90,1] + -4.250;
   1:  PR[GP1:91,2] = PR[GP1:90,2] + -15.315;
   1:L PR[91] 10mm/sec CNT100;
   1:  PR[GP1:91,1] = PR[GP1:90,1] + -2.360;
   1:  PR[GP1:91,2] = PR[GP1:90,2] + -13.193;
   1:L PR[91] 10mm/sec CNT100;
   1:  PR[GP1:91,1] = PR[GP1:90,1] + -1.099;
   1:  PR[GP1:91,2] = PR[GP1:90,2] + -12.456;
   1:L PR[91] 10mm/sec CNT100;
   1:  PR[GP1:91,1] = PR[GP1:90,1] + 1.979;
   1:  PR[GP1:91,2] = PR[GP1:90,2] + -12.426;
   1:L PR[91] 10mm/sec CNT100;
   1:  PR[GP1:91,1] = PR[GP1:90,1] + 3.606;
   1:  PR[GP1:91,2] = PR[GP1:90,2] + -14.375;
   1:L PR[91] 10mm/sec CNT100;
   1:  PR[GP1:91,1] = PR[GP1:90,1] + 4.566;
   1:  PR[GP1:91,2] = PR[GP1:90,2] + -14.980;
   1:L PR[91] 10mm/sec CNT100;
   1:  PR[GP1:91,1] = PR[GP1:90,1] + 5.007;
   1:  PR[GP1:91,2] = PR[GP1:90,2] + -15.221;
   1:L PR[91] 10mm/sec CNT100;
   1:  PR[GP1:91,1] = PR[GP1:90,1] + 8.227;
   1:  PR[GP1:91,2] = PR[GP1:90,2] + -19.628;
   1:L PR[91] 10mm/sec CNT100;
   1:  PR[GP1:91,1] = PR[GP1:90,1] + 10.905;
   1:  PR[GP1:91,2] = PR[GP1:90,2] + -23.510;
   1:L PR[91] 10mm/sec CNT100;
   1:  PR[GP1:91,1] = PR[GP1:90,1] + 11.645;
   1:  PR[GP1:91,2] = PR[GP1:90,2] + -24.227;
   1:L PR[91] 10mm/sec CNT100;
   1:  PR[GP1:91,1] = PR[GP1:90,1] + 18.731;
   1:  PR[GP1:91,2] = PR[GP1:90,2] + -29.704;
   1:L PR[91] 10mm/sec CNT100;
   1:  PR[GP1:91,1] = PR[GP1:90,1] + 21.899;
   1:  PR[GP1:91,2] = PR[GP1:90,2] + -31.249;
   1:L PR[91] 10mm/sec CNT100;
   1:  PR[GP1:91,1] = PR[GP1:90,1] + 28.159;
   1:  PR[GP1:91,2] = PR[GP1:90,2] + -33.625;
   1:L PR[91] 10mm/sec CNT100;
   1:  PR[GP1:91,1] = PR[GP1:90,1] + 34.266;
   1:  PR[GP1:91,2] = PR[GP1:90,2] + -34.524;
   1:L PR[91] 10mm/sec CNT100;
   1:  PR[GP1:91,1] = PR[GP1:90,1] + 38.561;
   1:  PR[GP1:91,2] = PR[GP1:90,2] + -34.831;
   1:L PR[91] 10mm/sec CNT100;
   1:  PR[GP1:91,1] = PR[GP1:90,1] + 47.033;
   1:  PR[GP1:91,2] = PR[GP1:90,2] + -33.466;
   1:L PR[91] 10mm/sec CNT100;
   1:  PR[GP1:91,1] = PR[GP1:90,1] + 49.097;
   1:  PR[GP1:91,2] = PR[GP1:90,2] + -33.003;
   1:L PR[91] 10mm/sec CNT100;
   1:  PR[GP1:91,1] = PR[GP1:90,1] + 58.458;
   1:  PR[GP1:91,2] = PR[GP1:90,2] + -28.303;
   1:L PR[91] 10mm/sec CNT100;
   1:  PR[GP1:91,1] = PR[GP1:90,1] + 58.778;
   1:  PR[GP1:91,2] = PR[GP1:90,2] + -28.123;
   1:L PR[91] 10mm/sec CNT100;
   1:  PR[GP1:91,1] = PR[GP1:90,1] + 66.544;
   1:  PR[GP1:91,2] = PR[GP1:90,2] + -20.479;
   1:L PR[91] 10mm/sec CNT100;
   1:  PR[GP1:91,1] = PR[GP1:90,1] + 66.838;
   1:  PR[GP1:91,2] = PR[GP1:90,2] + -19.941;
   1:L PR[91] 10mm/sec CNT100;
   1:  PR[GP1:91,1] = PR[GP1:90,1] + 71.564;
   1:  PR[GP1:91,2] = PR[GP1:90,2] + -10.821;
   1:L PR[91] 10mm/sec CNT100;
   1:  PR[GP1:91,1] = PR[GP1:90,1] + 71.781;
   1:  PR[GP1:91,2] = PR[GP1:90,2] + -9.540;
   1:L PR[91] 10mm/sec CNT100;
   1:  PR[GP1:91,1] = PR[GP1:90,1] + 73.307;
   1:  PR[GP1:91,2] = PR[GP1:90,2] + -0.007;
   1:L PR[91] 10mm/sec CNT100;
   1:  PR[GP1:91,1] = PR[GP1:90,1] + 73.057;
   1:  PR[GP1:91,2] = PR[GP1:90,2] + 1.468;
   1:L PR[91] 10mm/sec CNT100;
   1:  PR[GP1:91,1] = PR[GP1:90,1] + 71.563;
   1:  PR[GP1:91,2] = PR[GP1:90,2] + 10.815;
   1:L PR[91] 10mm/sec CNT100;
   1:  PR[GP1:91,1] = PR[GP1:90,1] + 66.838;
   1:  PR[GP1:91,2] = PR[GP1:90,2] + 19.932;
   1:L PR[91] 10mm/sec CNT100;
   1:  PR[GP1:91,1] = PR[GP1:90,1] + 66.544;
   1:  PR[GP1:91,2] = PR[GP1:90,2] + 20.470;
   1:L PR[91] 10mm/sec CNT100;
   1:  PR[GP1:91,1] = PR[GP1:90,1] + 58.778;
   1:  PR[GP1:91,2] = PR[GP1:90,2] + 28.115;
   1:L PR[91] 10mm/sec CNT100;
   1:  PR[GP1:91,1] = PR[GP1:90,1] + 58.458;
   1:  PR[GP1:91,2] = PR[GP1:90,2] + 28.295;
   1:L PR[91] 10mm/sec CNT100;
   1:  PR[GP1:91,1] = PR[GP1:90,1] + 49.097;
   1:  PR[GP1:91,2] = PR[GP1:90,2] + 32.994;
   1:L PR[91] 10mm/sec CNT100;
   1:  PR[GP1:91,1] = PR[GP1:90,1] + 47.033;
   1:  PR[GP1:91,2] = PR[GP1:90,2] + 33.457;
   1:L PR[91] 10mm/sec CNT100;
   1:  PR[GP1:91,1] = PR[GP1:90,1] + 38.561;
   1:  PR[GP1:91,2] = PR[GP1:90,2] + 34.822;
   1:L PR[91] 10mm/sec CNT100;
   1:  PR[GP1:91,1] = PR[GP1:90,1] + 34.266;
   1:  PR[GP1:91,2] = PR[GP1:90,2] + 34.516;
   1:L PR[91] 10mm/sec CNT100;
   1:  PR[GP1:91,1] = PR[GP1:90,1] + 28.159;
   1:  PR[GP1:91,2] = PR[GP1:90,2] + 33.617;
   1:L PR[91] 10mm/sec CNT100;
   1:  PR[GP1:91,1] = PR[GP1:90,1] + 21.899;
   1:  PR[GP1:91,2] = PR[GP1:90,2] + 31.240;
   1:L PR[91] 10mm/sec CNT100;
   1:  PR[GP1:91,1] = PR[GP1:90,1] + 18.731;
   1:  PR[GP1:91,2] = PR[GP1:90,2] + 29.695;
   1:L PR[91] 10mm/sec CNT100;
   1:  PR[GP1:91,1] = PR[GP1:90,1] + 11.645;
   1:  PR[GP1:91,2] = PR[GP1:90,2] + 24.218;
   1:L PR[91] 10mm/sec CNT100;
   1:  PR[GP1:91,1] = PR[GP1:90,1] + 10.904;
   1:  PR[GP1:91,2] = PR[GP1:90,2] + 23.501;
   1:L PR[91] 10mm/sec CNT100;
   1:  PR[GP1:91,1] = PR[GP1:90,1] + 8.173;
   1:  PR[GP1:91,2] = PR[GP1:90,2] + 19.544;
   1:L PR[91] 10mm/sec CNT100;
   1:  PR[GP1:91,1] = PR[GP1:90,1] + 5.067;
   1:  PR[GP1:91,2] = PR[GP1:90,2] + 15.295;
   1:L PR[91] 10mm/sec CNT100;
   1:  PR[GP1:91,1] = PR[GP1:90,1] + 3.122;
   1:  PR[GP1:91,2] = PR[GP1:90,2] + 13.154;
   1:L PR[91] 10mm/sec CNT100;
   1:  PR[GP1:91,1] = PR[GP1:90,1] + 1.860;
   1:  PR[GP1:91,2] = PR[GP1:90,2] + 12.418;
   1:L PR[91] 10mm/sec CNT100;
   1:  PR[GP1:91,1] = PR[GP1:90,1] + -0.873;
   1:  PR[GP1:91,2] = PR[GP1:90,2] + 13.366;
   1:  PR[GP1:91,3] = PR[GP1:90,3] + 31.920;
   1:L PR[91] 10mm/sec CNT100;
   1:  PR[GP1:91,1] = PR[GP1:90,1] + -2.622;
   1:  PR[GP1:91,2] = PR[GP1:90,2] + 14.390;
   1:L PR[91] 10mm/sec CNT100;
   1:  PR[GP1:91,1] = PR[GP1:90,1] + -4.272;
   1:  PR[GP1:91,2] = PR[GP1:90,2] + 16.170;
   1:L PR[91] 10mm/sec CNT100;
   1:  PR[GP1:91,1] = PR[GP1:90,1] + -4.284;
   1:  PR[GP1:91,2] = PR[GP1:90,2] + 16.280;
   1:L PR[91] 10mm/sec CNT100;
   1:  PR[GP1:91,1] = PR[GP1:90,1] + -9.521;
   1:  PR[GP1:91,2] = PR[GP1:90,2] + 23.440;
   1:L PR[91] 10mm/sec CNT100;
   1:  PR[GP1:91,1] = PR[GP1:90,1] + -9.889;
   1:  PR[GP1:91,2] = PR[GP1:90,2] + 23.871;
   1:L PR[91] 10mm/sec CNT100;
   1:  PR[GP1:91,1] = PR[GP1:90,1] + -13.098;
   1:  PR[GP1:91,2] = PR[GP1:90,2] + 26.245;
   1:L PR[91] 10mm/sec CNT100;
   1:  PR[GP1:91,1] = PR[GP1:90,1] + -18.074;
   1:  PR[GP1:91,2] = PR[GP1:90,2] + 30.087;
   1:L PR[91] 10mm/sec CNT100;
   1:  PR[GP1:91,1] = PR[GP1:90,1] + -19.425;
   1:  PR[GP1:91,2] = PR[GP1:90,2] + 30.746;
   1:L PR[91] 10mm/sec CNT100;
   1:  PR[GP1:91,1] = PR[GP1:90,1] + -27.487;
   1:  PR[GP1:91,2] = PR[GP1:90,2] + 33.810;
   1:L PR[91] 10mm/sec CNT100;
   1:  PR[GP1:91,1] = PR[GP1:90,1] + -31.709;
   1:  PR[GP1:91,2] = PR[GP1:90,2] + 34.430;
   1:L PR[91] 10mm/sec CNT100;
   1:  PR[GP1:91,1] = PR[GP1:90,1] + -37.822;
   1:  PR[GP1:91,2] = PR[GP1:90,2] + 34.864;
   1:L PR[91] 10mm/sec CNT100;
   1:  PR[GP1:91,1] = PR[GP1:90,1] + -44.544;
   1:  PR[GP1:91,2] = PR[GP1:90,2] + 33.781;
   1:L PR[91] 10mm/sec CNT100;
   1:  PR[GP1:91,1] = PR[GP1:90,1] + -48.267;
   1:  PR[GP1:91,2] = PR[GP1:90,2] + 32.948;
   1:L PR[91] 10mm/sec CNT100;
   1:  PR[GP1:91,1] = PR[GP1:90,1] + -56.166;
   1:  PR[GP1:91,2] = PR[GP1:90,2] + 28.975;
   1:L PR[91] 10mm/sec CNT100;
   1:  PR[GP1:91,1] = PR[GP1:90,1] + -57.854;
   1:  PR[GP1:91,2] = PR[GP1:90,2] + 28.023;
   1:L PR[91] 10mm/sec CNT100;
   1:  PR[GP1:91,1] = PR[GP1:90,1] + -65.161;
   1:  PR[GP1:91,2] = PR[GP1:90,2] + 20.855;
   1:L PR[91] 10mm/sec CNT100;
   1:  PR[GP1:91,1] = PR[GP1:90,1] + -65.591;
   1:  PR[GP1:91,2] = PR[GP1:90,2] + 20.402;
   1:L PR[91] 10mm/sec CNT100;
   1:  PR[GP1:91,1] = PR[GP1:90,1] + -70.620;
   1:  PR[GP1:91,2] = PR[GP1:90,2] + 10.742;
   1:L PR[91] 10mm/sec CNT100;
   1:  PR[GP1:91,1] = PR[GP1:90,1] + -72.342;
   1:  PR[GP1:91,2] = PR[GP1:90,2] + -0.002;
   1:L PR[91] 10mm/sec CNT100;
   1:  PR[GP1:91,1] = PR[GP1:90,1] + -72.308;
   1:  PR[GP1:91,2] = PR[GP1:90,2] + -0.200;
   1:L PR[91] 10mm/sec CNT100;
   1:  PR[GP1:91,1] = PR[GP1:90,1] + -70.620;
   1:  PR[GP1:91,2] = PR[GP1:90,2] + -10.751;
   1:L PR[91] 10mm/sec CNT100;
   1:  PR[GP1:91,1] = PR[GP1:90,1] + -65.591;
   1:  PR[GP1:91,2] = PR[GP1:90,2] + -20.411;
   1:L PR[91] 10mm/sec CNT100;
   1:  PR[GP1:91,1] = PR[GP1:90,1] + -65.161;
   1:  PR[GP1:91,2] = PR[GP1:90,2] + -20.863;
   1:L PR[91] 10mm/sec CNT100;
   1:  PR[GP1:91,1] = PR[GP1:90,1] + -57.854;
   1:  PR[GP1:91,2] = PR[GP1:90,2] + -28.032;
   1:L PR[91] 10mm/sec CNT100;
   1:  PR[GP1:91,1] = PR[GP1:90,1] + -56.166;
   1:  PR[GP1:91,2] = PR[GP1:90,2] + -28.984;
   1:L PR[91] 10mm/sec CNT100;
   1:  PR[GP1:91,1] = PR[GP1:90,1] + -48.267;
   1:  PR[GP1:91,2] = PR[GP1:90,2] + -32.956;
   1:L PR[91] 10mm/sec CNT100;
   1:  PR[GP1:91,1] = PR[GP1:90,1] + -44.545;
   1:  PR[GP1:91,2] = PR[GP1:90,2] + -33.790;
   1:L PR[91] 10mm/sec CNT100;
   1:  PR[GP1:91,1] = PR[GP1:90,1] + -37.822;
   1:  PR[GP1:91,2] = PR[GP1:90,2] + -34.873;
   1:L PR[91] 10mm/sec CNT100;
   1:  PR[GP1:91,1] = PR[GP1:90,1] + -31.709;
   1:  PR[GP1:91,2] = PR[GP1:90,2] + -34.438;
   1:L PR[91] 10mm/sec CNT100;
   1:  PR[GP1:91,1] = PR[GP1:90,1] + -27.487;
   1:  PR[GP1:91,2] = PR[GP1:90,2] + -33.819;
   1:L PR[91] 10mm/sec CNT100;
   1:  PR[GP1:91,1] = PR[GP1:90,1] + -19.425;
   1:  PR[GP1:91,2] = PR[GP1:90,2] + -30.754;
   1:L PR[91] 10mm/sec CNT100;
   1:  PR[GP1:91,1] = PR[GP1:90,1] + -18.074;
   1:  PR[GP1:91,2] = PR[GP1:90,2] + -30.096;
   1:L PR[91] 10mm/sec CNT100;
   1:  PR[GP1:91,1] = PR[GP1:90,1] + -13.097;
   1:  PR[GP1:91,2] = PR[GP1:90,2] + -26.253;
   1:L PR[91] 10mm/sec CNT100;
   1:  PR[GP1:91,1] = PR[GP1:90,1] + -10.216;
   1:  PR[GP1:91,2] = PR[GP1:90,2] + -24.143;
   1:L PR[91] 10mm/sec CNT100;
   1:  PR[GP1:91,1] = PR[GP1:90,1] + -9.896;
   1:  PR[GP1:91,2] = PR[GP1:90,2] + -23.888;
   1:L PR[91] 10mm/sec CNT100;
   1:  PR[GP1:91,1] = PR[GP1:90,1] + -9.521;
   1:  PR[GP1:91,2] = PR[GP1:90,2] + -23.449;
   1:L PR[91] 10mm/sec CNT100;
   1:  PR[GP1:91,1] = PR[GP1:90,1] + -4.173;
   1:  PR[GP1:91,2] = PR[GP1:90,2] + -16.136;
   1:L PR[91] 10mm/sec CNT100;
   1:  PR[GP1:91,1] = PR[GP1:90,1] + -2.627;
   1:  PR[GP1:91,2] = PR[GP1:90,2] + -14.401;
   1:L PR[91] 10mm/sec CNT100;
   1:  PR[GP1:91,1] = PR[GP1:90,1] + -0.873;
   1:  PR[GP1:91,2] = PR[GP1:90,2] + -13.375;
   1:L PR[91] 10mm/sec CNT100;
   1:  PR[GP1:91,1] = PR[GP1:90,1] + 1.764;
   1:  PR[GP1:91,2] = PR[GP1:90,2] + -13.350;
   1:L PR[91] 10mm/sec CNT100;
   1:  PR[GP1:91,1] = PR[GP1:90,1] + 3.139;
   1:  PR[GP1:91,2] = PR[GP1:90,2] + -14.997;
   1:L PR[91] 10mm/sec CNT100;
   1:  PR[GP1:91,1] = PR[GP1:90,1] + 3.923;
   1:  PR[GP1:91,2] = PR[GP1:90,2] + -15.491;
   1:L PR[91] 10mm/sec CNT100;
   1:  PR[GP1:91,1] = PR[GP1:90,1] + 4.933;
   1:  PR[GP1:91,2] = PR[GP1:90,2] + -16.044;
   1:L PR[91] 10mm/sec CNT100;
   1:  PR[GP1:91,1] = PR[GP1:90,1] + 10.343;
   1:  PR[GP1:91,2] = PR[GP1:90,2] + -23.446;
   1:L PR[91] 10mm/sec CNT100;
   1:  PR[GP1:91,1] = PR[GP1:90,1] + 10.714;
   1:  PR[GP1:91,2] = PR[GP1:90,2] + -23.880;
   1:L PR[91] 10mm/sec CNT100;
   1:  PR[GP1:91,1] = PR[GP1:90,1] + 13.919;
   1:  PR[GP1:91,2] = PR[GP1:90,2] + -26.253;
   1:L PR[91] 10mm/sec CNT100;
   1:  PR[GP1:91,1] = PR[GP1:90,1] + 18.893;
   1:  PR[GP1:91,2] = PR[GP1:90,2] + -30.098;
   1:L PR[91] 10mm/sec CNT100;
   1:  PR[GP1:91,1] = PR[GP1:90,1] + 20.243;
   1:  PR[GP1:91,2] = PR[GP1:90,2] + -30.756;
   1:L PR[91] 10mm/sec CNT100;
   1:  PR[GP1:91,1] = PR[GP1:90,1] + 28.304;
   1:  PR[GP1:91,2] = PR[GP1:90,2] + -33.816;
   1:L PR[91] 10mm/sec CNT100;
   1:  PR[GP1:91,1] = PR[GP1:90,1] + 32.525;
   1:  PR[GP1:91,2] = PR[GP1:90,2] + -34.438;
   1:L PR[91] 10mm/sec CNT100;
   1:  PR[GP1:91,1] = PR[GP1:90,1] + 38.637;
   1:  PR[GP1:91,2] = PR[GP1:90,2] + -34.874;
   1:L PR[91] 10mm/sec CNT100;
   1:  PR[GP1:91,1] = PR[GP1:90,1] + 45.359;
   1:  PR[GP1:91,2] = PR[GP1:90,2] + -33.791;
   1:L PR[91] 10mm/sec CNT100;
   1:  PR[GP1:91,1] = PR[GP1:90,1] + 49.082;
   1:  PR[GP1:91,2] = PR[GP1:90,2] + -32.956;
   1:L PR[91] 10mm/sec CNT100;
   1:  PR[GP1:91,1] = PR[GP1:90,1] + 56.982;
   1:  PR[GP1:91,2] = PR[GP1:90,2] + -28.990;
   1:L PR[91] 10mm/sec CNT100;
   1:  PR[GP1:91,1] = PR[GP1:90,1] + 58.670;
   1:  PR[GP1:91,2] = PR[GP1:90,2] + -28.040;
   1:L PR[91] 10mm/sec CNT100;
   1:  PR[GP1:91,1] = PR[GP1:90,1] + 65.978;
   1:  PR[GP1:91,2] = PR[GP1:90,2] + -20.859;
   1:L PR[91] 10mm/sec CNT100;
   1:  PR[GP1:91,1] = PR[GP1:90,1] + 66.409;
   1:  PR[GP1:91,2] = PR[GP1:90,2] + -20.405;
   1:L PR[91] 10mm/sec CNT100;
   1:  PR[GP1:91,1] = PR[GP1:90,1] + 71.439;
   1:  PR[GP1:91,2] = PR[GP1:90,2] + -10.769;
   1:L PR[91] 10mm/sec CNT100;
   1:  PR[GP1:91,1] = PR[GP1:90,1] + 73.163;
   1:  PR[GP1:91,2] = PR[GP1:90,2] + -0.004;
   1:L PR[91] 10mm/sec CNT100;
   1:  PR[GP1:91,1] = PR[GP1:90,1] + 71.439;
   1:  PR[GP1:91,2] = PR[GP1:90,2] + 10.760;
   1:L PR[91] 10mm/sec CNT100;
   1:  PR[GP1:91,1] = PR[GP1:90,1] + 66.409;
   1:  PR[GP1:91,2] = PR[GP1:90,2] + 20.396;
   1:L PR[91] 10mm/sec CNT100;
   1:  PR[GP1:91,1] = PR[GP1:90,1] + 65.978;
   1:  PR[GP1:91,2] = PR[GP1:90,2] + 20.851;
   1:L PR[91] 10mm/sec CNT100;
   1:  PR[GP1:91,1] = PR[GP1:90,1] + 58.670;
   1:  PR[GP1:91,2] = PR[GP1:90,2] + 28.031;
   1:L PR[91] 10mm/sec CNT100;
   1:  PR[GP1:91,1] = PR[GP1:90,1] + 56.982;
   1:  PR[GP1:91,2] = PR[GP1:90,2] + 28.981;
   1:L PR[91] 10mm/sec CNT100;
   1:  PR[GP1:91,1] = PR[GP1:90,1] + 49.082;
   1:  PR[GP1:91,2] = PR[GP1:90,2] + 32.947;
   1:L PR[91] 10mm/sec CNT100;
   1:  PR[GP1:91,1] = PR[GP1:90,1] + 45.359;
   1:  PR[GP1:91,2] = PR[GP1:90,2] + 33.782;
   1:L PR[91] 10mm/sec CNT100;
   1:  PR[GP1:91,1] = PR[GP1:90,1] + 38.637;
   1:  PR[GP1:91,2] = PR[GP1:90,2] + 34.865;
   1:L PR[91] 10mm/sec CNT100;
   1:  PR[GP1:91,1] = PR[GP1:90,1] + 32.525;
   1:  PR[GP1:91,2] = PR[GP1:90,2] + 34.429;
   1:L PR[91] 10mm/sec CNT100;
   1:  PR[GP1:91,1] = PR[GP1:90,1] + 28.304;
   1:  PR[GP1:91,2] = PR[GP1:90,2] + 33.807;
   1:L PR[91] 10mm/sec CNT100;
   1:  PR[GP1:91,1] = PR[GP1:90,1] + 20.243;
   1:  PR[GP1:91,2] = PR[GP1:90,2] + 30.748;
   1:L PR[91] 10mm/sec CNT100;
   1:  PR[GP1:91,1] = PR[GP1:90,1] + 18.893;
   1:  PR[GP1:91,2] = PR[GP1:90,2] + 30.089;
   1:L PR[91] 10mm/sec CNT100;
   1:  PR[GP1:91,1] = PR[GP1:90,1] + 13.918;
   1:  PR[GP1:91,2] = PR[GP1:90,2] + 26.244;
   1:L PR[91] 10mm/sec CNT100;
   1:  PR[GP1:91,1] = PR[GP1:90,1] + 11.038;
   1:  PR[GP1:91,2] = PR[GP1:90,2] + 24.132;
   1:L PR[91] 10mm/sec CNT100;
   1:  PR[GP1:91,1] = PR[GP1:90,1] + 10.721;
   1:  PR[GP1:91,2] = PR[GP1:90,2] + 23.880;
   1:L PR[91] 10mm/sec CNT100;
   1:  PR[GP1:91,1] = PR[GP1:90,1] + 10.343;
   1:  PR[GP1:91,2] = PR[GP1:90,2] + 23.438;
   1:L PR[91] 10mm/sec CNT100;
   1:  PR[GP1:91,1] = PR[GP1:90,1] + 4.993;
   1:  PR[GP1:91,2] = PR[GP1:90,2] + 16.118;
   1:L PR[91] 10mm/sec CNT100;
   1:  PR[GP1:91,1] = PR[GP1:90,1] + 3.403;
   1:  PR[GP1:91,2] = PR[GP1:90,2] + 14.367;
   1:L PR[91] 10mm/sec CNT100;
   1:  PR[GP1:91,1] = PR[GP1:90,1] + 1.645;
   1:  PR[GP1:91,2] = PR[GP1:90,2] + 13.342;
   1:L PR[91] 10mm/sec CNT100;
   1:  PR[GP1:91,1] = PR[GP1:90,1] + -0.647;
   1:  PR[GP1:91,2] = PR[GP1:90,2] + 14.286;
   1:  PR[GP1:91,3] = PR[GP1:90,3] + 33.250;
   1:L PR[91] 10mm/sec CNT100;
   1:  PR[GP1:91,1] = PR[GP1:90,1] + -2.890;
   1:  PR[GP1:91,2] = PR[GP1:90,2] + 15.598;
   1:L PR[91] 10mm/sec CNT100;
   1:  PR[GP1:91,1] = PR[GP1:90,1] + -4.197;
   1:  PR[GP1:91,2] = PR[GP1:90,2] + 17.008;
   1:L PR[91] 10mm/sec CNT100;
   1:  PR[GP1:91,1] = PR[GP1:90,1] + -4.207;
   1:  PR[GP1:91,2] = PR[GP1:90,2] + 17.101;
   1:L PR[91] 10mm/sec CNT100;
   1:  PR[GP1:91,1] = PR[GP1:90,1] + -8.184;
   1:  PR[GP1:91,2] = PR[GP1:90,2] + 22.539;
   1:L PR[91] 10mm/sec CNT100;
   1:  PR[GP1:91,1] = PR[GP1:90,1] + -9.464;
   1:  PR[GP1:91,2] = PR[GP1:90,2] + 24.037;
   1:L PR[91] 10mm/sec CNT100;
   1:  PR[GP1:91,1] = PR[GP1:90,1] + -17.972;
   1:  PR[GP1:91,2] = PR[GP1:90,2] + 30.342;
   1:L PR[91] 10mm/sec CNT100;
   1:  PR[GP1:91,1] = PR[GP1:90,1] + -18.119;
   1:  PR[GP1:91,2] = PR[GP1:90,2] + 30.423;
